LIN {X 0,Y 496.751,Z 364.923,A -85,B 0,C 180,E1 23860.178,E2 23860.178} C_VEL
LIN {X 0,Y 496.699,Z 364.922,A -85,B 0,C 180,E1 23856.821,E2 23856.821} C_VEL
LIN {X 0,Y 496.696,Z 364.92,A -85,B 0,C 180,E1 23853.178,E2 23853.178} C_VEL
LIN {X 0,Y 496.745,Z 364.921,A -85,B 0,C 180,E1 23849.769,E2 23849.769} C_VEL
LIN {X 0,Y 496.722,Z 364.92,A -85,B 0,C 180,E1 23846.307,E2 23846.307} C_VEL
LIN {X 0,Y 496.696,Z 364.92,A -85,B 0,C 180,E1 23842.943,E2 23842.943} C_VEL
LIN {X 0,Y 496.732,Z 364.923,A -85,B 0,C 180,E1 23839.563,E2 23839.563} C_VEL
LIN {X 0,Y 496.727,Z 364.921,A -85,B 0,C 180,E1 23836.141,E2 23836.141} C_VEL
LIN {X 0,Y 496.694,Z 364.922,A -85,B 0,C 180,E1 23832.787,E2 23832.787} C_VEL
LIN {X 0,Y 496.723,Z 364.923,A -85,B 0,C 180,E1 23829.374,E2 23829.374} C_VEL
LIN {X 0,Y 496.725,Z 364.922,A -85,B 0,C 180,E1 23826.045,E2 23826.045} C_VEL
LIN {X 0,Y 496.693,Z 364.922,A -85,B 0,C 180,E1 23822.592,E2 23822.592} C_VEL
LIN {X 0,Y 496.711,Z 364.924,A -85,B 0,C 180,E1 23819.116,E2 23819.116} C_VEL
LIN {X 0,Y 496.752,Z 364.924,A -85,B 0,C 180,E1 23815.696,E2 23815.696} C_VEL
LIN {X 0,Y 496.697,Z 364.925,A -85,B 0,C 180,E1 23812.269,E2 23812.269} C_VEL
LIN {X 0,Y 496.694,Z 364.923,A -85,B 0,C 180,E1 23808.679,E2 23808.679} C_VEL
LIN {X 0,Y 496.739,Z 364.924,A -85,B 0,C 180,E1 23805.279,E2 23805.279} C_VEL
LIN {X 0,Y 496.717,Z 364.924,A -85,B 0,C 180,E1 23801.859,E2 23801.859} C_VEL
LIN {X 0,Y 496.691,Z 364.925,A -85,B 0,C 180,E1 23798.457,E2 23798.457} C_VEL
LIN {X 0,Y 496.723,Z 364.926,A -85,B 0,C 180,E1 23795.007,E2 23795.007} C_VEL
LIN {X 0,Y 496.737,Z 364.925,A -85,B 0,C 180,E1 23791.557,E2 23791.557} C_VEL
LIN {X 0,Y 496.735,Z 365.024,A -85,B 0,C 180,E1 23790.965,E2 23790.965} C_VEL
LIN {X 0,Y 501.684,Z 383.717,A -85,B 0,C 180,E1 23788.187,E2 23788.187} C_VEL
LIN {X 0,Y 500.546,Z 410.556,A -85,B 0,C 180,E1 23784.802,E2 23784.802} C_VEL
LIN {X 0,Y 499.492,Z 438.729,A -85,B 0,C 180,E1 23781.304,E2 23781.304} C_VEL
LIN {X 0,Y 498.454,Z 468.768,A -85,B 0,C 180,E1 23777.632,E2 23777.632} C_VEL
LIN {X 0,Y 498.176,Z 480.291,A -85,B 0,C 180,E1 23776.272,E2 23776.272} C_VEL
LIN {X 0,Y 499.98,Z 493.845,A -85,B 0,C 180,E1 23775.974,E2 23775.974} C_VEL
LIN {X 0,Y 498.863,Z 596.511,A -85,B 0,C 180,E1 23774.304,E2 23774.304} C_VEL
LIN {X 0,Y 498.66,Z 611.149,A -85,B 0,C 180,E1 23773.864,E2 23773.864} C_VEL
LIN {X 0,Y 498.343,Z 626.502,A -85,B 0,C 180,E1 23773.163,E2 23773.163} C_VEL
LIN {X 0,Y 497.924,Z 640.34,A -85,B 0,C 180,E1 23772.29,E2 23772.29} C_VEL
LIN {X 0,Y 497.546,Z 652.64,A -85,B 0,C 180,E1 23771.28,E2 23771.28} C_VEL
LIN {X 0,Y 497.197,Z 664.163,A -85,B 0,C 180,E1 23770.076,E2 23770.076} C_VEL
LIN {X 0,Y 496.862,Z 674.559,A -85,B 0,C 180,E1 23768.681,E2 23768.681} C_VEL
LIN {X 0,Y 496.633,Z 682.68,A -85,B 0,C 180,E1 23767.287,E2 23767.287} C_VEL
LIN {X 0,Y 496.463,Z 689.464,A -85,B 0,C 180,E1 23765.78,E2 23765.78} C_VEL
LIN {X 0,Y 496.36,Z 694.745,A -85,B 0,C 180,E1 23764.159,E2 23764.159} C_VEL
LIN {X 0,Y 496.314,Z 698.292,A -85,B 0,C 180,E1 23762.54,E2 23762.54} C_VEL
LIN {X 0,Y 496.314,Z 700.303,A -85,B 0,C 180,E1 23760.693,E2 23760.693} C_VEL
LIN {X 0,Y 496.325,Z 700.295,A -85,B 0,C 180,E1 23758.961,E2 23758.961} C_VEL
LIN {X 0,Y 496.378,Z 698.701,A -85,B 0,C 180,E1 23757.345,E2 23757.345} C_VEL
LIN {X 0,Y 496.477,Z 695.115,A -85,B 0,C 180,E1 23755.611,E2 23755.611} C_VEL
LIN {X 0,Y 496.626,Z 689.899,A -85,B 0,C 180,E1 23753.991,E2 23753.991} C_VEL
LIN {X 0,Y 496.84,Z 683.239,A -85,B 0,C 180,E1 23752.484,E2 23752.484} C_VEL
LIN {X 0,Y 497.137,Z 674.143,A -85,B 0,C 180,E1 23750.94,E2 23750.94} C_VEL
LIN {X 0,Y 497.497,Z 664.083,A -85,B 0,C 180,E1 23749.62,E2 23749.62} C_VEL
LIN {X 0,Y 497.881,Z 653.043,A -85,B 0,C 180,E1 23748.474,E2 23748.474} C_VEL
LIN {X 0,Y 498.288,Z 640.076,A -85,B 0,C 180,E1 23747.425,E2 23747.425} C_VEL
LIN {X 0,Y 498.681,Z 626.863,A -85,B 0,C 180,E1 23746.61,E2 23746.61} C_VEL
LIN {X 0,Y 499.001,Z 612.986,A -85,B 0,C 180,E1 23745.969,E2 23745.969} C_VEL
LIN {X 0,Y 499.261,Z 596.561,A -85,B 0,C 180,E1 23745.466,E2 23745.466} C_VEL
LIN {X 0,Y 501.106,Z 491.5,A -85,B 0,C 180,E1 23743.486,E2 23743.486} C_VEL
LIN {X 0,Y 498.994,Z 479.897,A -85,B 0,C 180,E1 23743.11,E2 23743.11} C_VEL
LIN {X 0,Y 500.287,Z 449.814,A -85,B 0,C 180,E1 23739.345,E2 23739.345} C_VEL
LIN {X 0,Y 501.876,Z 420.998,A -85,B 0,C 180,E1 23735.645,E2 23735.645} C_VEL
LIN {X 0,Y 503.631,Z 394.385,A -85,B 0,C 180,E1 23732.125,E2 23732.125} C_VEL
LIN {X 0,Y 503.952,Z 388.255,A -85,B 0,C 180,E1 23731.277,E2 23731.277} C_VEL
LIN {X 0,Y 500.616,Z 376.388,A -85,B 0,C 180,E1 23729.185,E2 23729.185} C_VEL
LIN {X 0,Y 497.744,Z 368.01,A -85,B 0,C 180,E1 23727.532,E2 23727.532} C_VEL
LIN {X 0,Y 496.733,Z 364.926,A -85,B 0,C 180,E1 23726.862,E2 23726.862} C_VEL
LIN {X 0,Y 496.695,Z 364.928,A -85,B 0,C 180,E1 23723.426,E2 23723.426} C_VEL
LIN {X 0,Y 496.705,Z 364.927,A -85,B 0,C 180,E1 23719.898,E2 23719.898} C_VEL
LIN {X 0,Y 496.754,Z 364.923,A -85,B 0,C 180,E1 23716.499,E2 23716.499} C_VEL
LIN {X 0,Y 496.707,Z 364.927,A -85,B 0,C 180,E1 23713.032,E2 23713.032} C_VEL
LIN {X 0,Y 496.698,Z 364.929,A -85,B 0,C 180,E1 23709.558,E2 23709.558} C_VEL
LIN {X 0,Y 496.731,Z 364.976,A -85,B 0,C 180,E1 23706.762,E2 23706.762} C_VEL
LIN {X 0,Y 501.559,Z 377.294,A -85,B 0,C 180,E1 23704.76,E2 23704.76} C_VEL
LIN {X 0,Y 505.972,Z 390.476,A -85,B 0,C 180,E1 23702.98,E2 23702.98} C_VEL
LIN {X 0,Y 506.201,Z 393.068,A -85,B 0,C 180,E1 23702.707,E2 23702.707} C_VEL
LIN {X 0,Y 503.796,Z 428.513,A -85,B 0,C 180,E1 23699.616,E2 23699.616} C_VEL
LIN {X 0,Y 502.352,Z 459.871,A -85,B 0,C 180,E1 23697.072,E2 23697.072} C_VEL
LIN {X 0,Y 504.653,Z 479.011,A -85,B 0,C 180,E1 23696.617,E2 23696.617} C_VEL
LIN {X 0,Y 502.285,Z 671.543,A -85,B 0,C 180,E1 23693.566,E2 23693.566} C_VEL
LIN {X 0,Y 501.774,Z 690.29,A -85,B 0,C 180,E1 23693.063,E2 23693.063} C_VEL
LIN {X 0,Y 501.171,Z 707.716,A -85,B 0,C 180,E1 23692.399,E2 23692.399} C_VEL
LIN {X 0,Y 500.457,Z 725.455,A -85,B 0,C 180,E1 23691.507,E2 23691.507} C_VEL
LIN {X 0,Y 499.694,Z 742.452,A -85,B 0,C 180,E1 23690.425,E2 23690.425} C_VEL
LIN {X 0,Y 498.903,Z 758.968,A -85,B 0,C 180,E1 23689.128,E2 23689.128} C_VEL
LIN {X 0,Y 498.093,Z 776.364,A -85,B 0,C 180,E1 23687.464,E2 23687.464} C_VEL
LIN {X 0,Y 497.466,Z 790.207,A -85,B 0,C 180,E1 23685.864,E2 23685.864} C_VEL
LIN {X 0,Y 496.95,Z 802.925,A -85,B 0,C 180,E1 23684.09,E2 23684.09} C_VEL
LIN {X 0,Y 496.554,Z 814.06,A -85,B 0,C 180,E1 23682.206,E2 23682.206} C_VEL
LIN {X 0,Y 496.27,Z 823.123,A -85,B 0,C 180,E1 23680.33,E2 23680.33} C_VEL
LIN {X 0,Y 496.103,Z 830.766,A -85,B 0,C 180,E1 23678.344,E2 23678.344} C_VEL
LIN {X 0,Y 495.998,Z 836.603,A -85,B 0,C 180,E1 23676.366,E2 23676.366} C_VEL
LIN {X 0,Y 495.942,Z 840.96,A -85,B 0,C 180,E1 23674.278,E2 23674.278} C_VEL
LIN {X 0,Y 495.928,Z 843.567,A -85,B 0,C 180,E1 23672.195,E2 23672.195} C_VEL
LIN {X 0,Y 495.93,Z 844.497,A -85,B 0,C 180,E1 23670,E2 23670} C_VEL
LIN {X 0,Y 495.928,Z 843.574,A -85,B 0,C 180,E1 23667.805,E2 23667.805} C_VEL
LIN {X 0,Y 495.94,Z 840.986,A -85,B 0,C 180,E1 23665.722,E2 23665.722} C_VEL
LIN {X 0,Y 495.994,Z 836.643,A -85,B 0,C 180,E1 23663.628,E2 23663.628} C_VEL
LIN {X 0,Y 496.101,Z 830.493,A -85,B 0,C 180,E1 23661.539,E2 23661.539} C_VEL
LIN {X 0,Y 496.28,Z 822.486,A -85,B 0,C 180,E1 23659.475,E2 23659.475} C_VEL
LIN {X 0,Y 496.582,Z 813.139,A -85,B 0,C 180,E1 23657.558,E2 23657.558} C_VEL
LIN {X 0,Y 497.007,Z 801.856,A -85,B 0,C 180,E1 23655.673,E2 23655.673} C_VEL
LIN {X 0,Y 497.572,Z 788.991,A -85,B 0,C 180,E1 23653.9,E2 23653.9} C_VEL
LIN {X 0,Y 498.237,Z 775.03,A -85,B 0,C 180,E1 23652.3,E2 23652.3} C_VEL
LIN {X 0,Y 498.965,Z 760.111,A -85,B 0,C 180,E1 23650.875,E2 23650.875} C_VEL
LIN {X 0,Y 499.76,Z 743.736,A -85,B 0,C 180,E1 23649.583,E2 23649.583} C_VEL
LIN {X 0,Y 500.53,Z 726.786,A -85,B 0,C 180,E1 23648.496,E2 23648.496} C_VEL
LIN {X 0,Y 501.249,Z 709.283,A -85,B 0,C 180,E1 23647.605,E2 23647.605} C_VEL
LIN {X 0,Y 501.911,Z 690.523,A -85,B 0,C 180,E1 23646.882,E2 23646.882} C_VEL
LIN {X 0,Y 502.427,Z 671.773,A -85,B 0,C 180,E1 23646.379,E2 23646.379} C_VEL
LIN {X 0,Y 502.791,Z 638.461,A -85,B 0,C 180,E1 23645.851,E2 23645.851} C_VEL
LIN {X 0,Y 504.288,Z 488.771,A -85,B 0,C 180,E1 23643.587,E2 23643.587} C_VEL
LIN {X 0,Y 504.3,Z 475.833,A -85,B 0,C 180,E1 23643.348,E2 23643.348} C_VEL
LIN {X 0,Y 502.499,Z 461.039,A -85,B 0,C 180,E1 23642.946,E2 23642.946} C_VEL
LIN {X 0,Y 504.592,Z 415.262,A -85,B 0,C 180,E1 23639.254,E2 23639.254} C_VEL
LIN {X 0,Y 505.68,Z 390.578,A -85,B 0,C 180,E1 23637.196,E2 23637.196} C_VEL
LIN {X 0,Y 497.568,Z 367.691,A -85,B 0,C 180,E1 23634.572,E2 23634.572} C_VEL
LIN {X 0,Y 496.708,Z 364.925,A -85,B 0,C 180,E1 23634.216,E2 23634.216} C_VEL
LIN {X 0,Y 496.698,Z 364.926,A -85,B 0,C 180,E1 23630.796,E2 23630.796} C_VEL
LIN {X 0,Y 496.75,Z 364.923,A -85,B 0,C 180,E1 23627.444,E2 23627.444} C_VEL
LIN {X 0,Y 496.717,Z 364.926,A -85,B 0,C 180,E1 23623.984,E2 23623.984} C_VEL
LIN {X 0,Y 496.693,Z 364.926,A -85,B 0,C 180,E1 23620.557,E2 23620.557} C_VEL
LIN {X 0,Y 496.729,Z 364.926,A -85,B 0,C 180,E1 23617.145,E2 23617.145} C_VEL
LIN {X 0,Y 496.725,Z 364.928,A -85,B 0,C 180,E1 23613.749,E2 23613.749} C_VEL
LIN {X 0,Y 496.733,Z 365.09,A -85,B 0,C 180,E1 23611.877,E2 23611.877} C_VEL
LIN {X 0,Y 502.332,Z 381.373,A -85,B 0,C 180,E1 23609.918,E2 23609.918} C_VEL
LIN {X 0,Y 504.151,Z 388.316,A -85,B 0,C 180,E1 23609.136,E2 23609.136} C_VEL
LIN {X 0,Y 503.782,Z 409.778,A -85,B 0,C 180,E1 23607.21,E2 23607.21} C_VEL
LIN {X 0,Y 505.798,Z 422.143,A -85,B 0,C 180,E1 23606.837,E2 23606.837} C_VEL
LIN {X 0,Y 503.551,Z 543.564,A -85,B 0,C 180,E1 23604.775,E2 23604.775} C_VEL
LIN {X 0,Y 502.661,Z 617.661,A -85,B 0,C 180,E1 23603.578,E2 23603.578} C_VEL
LIN {X 0,Y 502.231,Z 637.007,A -85,B 0,C 180,E1 23603.045,E2 23603.045} C_VEL
LIN {X 0,Y 501.643,Z 655.449,A -85,B 0,C 180,E1 23602.315,E2 23602.315} C_VEL
LIN {X 0,Y 500.959,Z 672.625,A -85,B 0,C 180,E1 23601.423,E2 23601.423} C_VEL
LIN {X 0,Y 500.205,Z 689.014,A -85,B 0,C 180,E1 23600.353,E2 23600.353} C_VEL
LIN {X 0,Y 499.419,Z 704.671,A -85,B 0,C 180,E1 23599.096,E2 23599.096} C_VEL
LIN {X 0,Y 498.61,Z 719.701,A -85,B 0,C 180,E1 23597.626,E2 23597.626} C_VEL
LIN {X 0,Y 497.909,Z 732.715,A -85,B 0,C 180,E1 23596.088,E2 23596.088} C_VEL
LIN {X 0,Y 497.261,Z 745.111,A -85,B 0,C 180,E1 23594.319,E2 23594.319} C_VEL
LIN {X 0,Y 496.775,Z 755.393,A -85,B 0,C 180,E1 23592.535,E2 23592.535} C_VEL
LIN {X 0,Y 496.395,Z 764.643,A -85,B 0,C 180,E1 23590.562,E2 23590.562} C_VEL
LIN {X 0,Y 496.155,Z 772.012,A -85,B 0,C 180,E1 23588.576,E2 23588.576} C_VEL
LIN {X 0,Y 496.012,Z 777.934,A -85,B 0,C 180,E1 23586.481,E2 23586.481} C_VEL
LIN {X 0,Y 495.949,Z 782.094,A -85,B 0,C 180,E1 23584.394,E2 23584.394} C_VEL
LIN {X 0,Y 495.931,Z 784.724,A -85,B 0,C 180,E1 23582.195,E2 23582.195} C_VEL
LIN {X 0,Y 495.93,Z 785.607,A -85,B 0,C 180,E1 23580,E2 23580} C_VEL
LIN {X 0,Y 495.927,Z 784.755,A -85,B 0,C 180,E1 23577.805,E2 23577.805} C_VEL
LIN {X 0,Y 495.946,Z 782.175,A -85,B 0,C 180,E1 23575.606,E2 23575.606} C_VEL
LIN {X 0,Y 496.007,Z 778.067,A -85,B 0,C 180,E1 23573.518,E2 23573.518} C_VEL
LIN {X 0,Y 496.138,Z 772.194,A -85,B 0,C 180,E1 23571.423,E2 23571.423} C_VEL
LIN {X 0,Y 496.368,Z 764.816,A -85,B 0,C 180,E1 23569.423,E2 23569.423} C_VEL
LIN {X 0,Y 496.738,Z 755.595,A -85,B 0,C 180,E1 23567.444,E2 23567.444} C_VEL
LIN {X 0,Y 497.252,Z 744.768,A -85,B 0,C 180,E1 23565.562,E2 23565.562} C_VEL
LIN {X 0,Y 497.909,Z 732.382,A -85,B 0,C 180,E1 23563.792,E2 23563.792} C_VEL
LIN {X 0,Y 498.693,Z 718.34,A -85,B 0,C 180,E1 23562.136,E2 23562.136} C_VEL
LIN {X 0,Y 499.508,Z 703.773,A -85,B 0,C 180,E1 23560.714,E2 23560.714} C_VEL
LIN {X 0,Y 500.33,Z 688.341,A -85,B 0,C 180,E1 23559.468,E2 23559.468} C_VEL
LIN {X 0,Y 501.139,Z 672.097,A -85,B 0,C 180,E1 23558.397,E2 23558.397} C_VEL
LIN {X 0,Y 501.883,Z 655.312,A -85,B 0,C 180,E1 23557.511,E2 23557.511} C_VEL
LIN {X 0,Y 502.537,Z 636.894,A -85,B 0,C 180,E1 23556.765,E2 23556.765} C_VEL
LIN {X 0,Y 503.041,Z 617.958,A -85,B 0,C 180,E1 23556.222,E2 23556.222} C_VEL
LIN {X 0,Y 503.395,Z 592.619,A -85,B 0,C 180,E1 23555.783,E2 23555.783} C_VEL
LIN {X 0,Y 505.661,Z 420.696,A -85,B 0,C 180,E1 23553.073,E2 23553.073} C_VEL
LIN {X 0,Y 504.059,Z 412.019,A -85,B 0,C 180,E1 23552.83,E2 23552.83} C_VEL
LIN {X 0,Y 503.132,Z 407.014,A -85,B 0,C 180,E1 23552.598,E2 23552.598} C_VEL
LIN {X 0,Y 501.689,Z 400.932,A -85,B 0,C 180,E1 23552.074,E2 23552.074} C_VEL
LIN {X 0,Y 498.85,Z 394.215,A -85,B 0,C 180,E1 23551.252,E2 23551.252} C_VEL
LIN {X 0,Y 495.123,Z 386.112,A -85,B 0,C 180,E1 23550.212,E2 23550.212} C_VEL
LIN {X 0,Y 488.761,Z 365.913,A -85,B 0,C 180,E1 23547.763,E2 23547.763} C_VEL
LIN {X 0,Y 488.803,Z 365.91,A -85,B 0,C 180,E1 23544.34,E2 23544.34} C_VEL
LIN {X 0,Y 488.793,Z 365.913,A -85,B 0,C 180,E1 23540.83,E2 23540.83} C_VEL
LIN {X 0,Y 488.759,Z 365.913,A -85,B 0,C 180,E1 23537.38,E2 23537.38} C_VEL
LIN {X 0,Y 488.776,Z 365.913,A -85,B 0,C 180,E1 23533.906,E2 23533.906} C_VEL
LIN {X 0,Y 488.826,Z 365.911,A -85,B 0,C 180,E1 23530.422,E2 23530.422} C_VEL
LIN {X 0,Y 488.769,Z 365.912,A -85,B 0,C 180,E1 23526.972,E2 23526.972} C_VEL
LIN {X 0,Y 488.758,Z 365.913,A -85,B 0,C 180,E1 23523.388,E2 23523.388} C_VEL
LIN {X 0,Y 488.789,Z 365.911,A -85,B 0,C 180,E1 23519.942,E2 23519.942} C_VEL
LIN {X 0,Y 488.8,Z 365.911,A -85,B 0,C 180,E1 23516.483,E2 23516.483} C_VEL
LIN {X 0,Y 488.758,Z 365.911,A -85,B 0,C 180,E1 23513.128,E2 23513.128} C_VEL
LIN {X 0,Y 488.771,Z 365.912,A -85,B 0,C 180,E1 23509.602,E2 23509.602} C_VEL
LIN {X 0,Y 488.818,Z 365.91,A -85,B 0,C 180,E1 23506.152,E2 23506.152} C_VEL
LIN {X 0,Y 488.764,Z 365.909,A -85,B 0,C 180,E1 23502.764,E2 23502.764} C_VEL
LIN {X 0,Y 488.758,Z 365.909,A -85,B 0,C 180,E1 23499.182,E2 23499.182} C_VEL
LIN {X 0,Y 488.795,Z 365.911,A -85,B 0,C 180,E1 23495.753,E2 23495.753} C_VEL
LIN {X 0,Y 488.798,Z 365.908,A -85,B 0,C 180,E1 23492.227,E2 23492.227} C_VEL
LIN {X 0,Y 488.755,Z 365.909,A -85,B 0,C 180,E1 23488.828,E2 23488.828} C_VEL
LIN {X 0,Y 488.766,Z 365.912,A -85,B 0,C 180,E1 23485.306,E2 23485.306} C_VEL
LIN {X 0,Y 488.82,Z 365.908,A -85,B 0,C 180,E1 23481.886,E2 23481.886} C_VEL
LIN {X 0,Y 488.767,Z 365.911,A -85,B 0,C 180,E1 23478.435,E2 23478.435} C_VEL
LIN {X 0,Y 488.757,Z 365.912,A -85,B 0,C 180,E1 23474.924,E2 23474.924} C_VEL
LIN {X 0,Y 488.798,Z 365.913,A -85,B 0,C 180,E1 23471.515,E2 23471.515} C_VEL
LIN {X 0,Y 488.792,Z 365.911,A -85,B 0,C 180,E1 23468.016,E2 23468.016} C_VEL
LIN {X 0,Y 488.756,Z 365.911,A -85,B 0,C 180,E1 23464.558,E2 23464.558} C_VEL
LIN {X 0,Y 488.764,Z 365.911,A -85,B 0,C 180,E1 23460.999,E2 23460.999} C_VEL
LIN {X 0,Y 488.815,Z 365.913,A -85,B 0,C 180,E1 23457.594,E2 23457.594} C_VEL
LIN {X 0,Y 488.769,Z 365.914,A -85,B 0,C 180,E1 23454.105,E2 23454.105} C_VEL
LIN {X 0,Y 488.754,Z 365.914,A -85,B 0,C 180,E1 23450.641,E2 23450.641} C_VEL
LIN {X 0,Y 488.792,Z 365.913,A -85,B 0,C 180,E1 23447.224,E2 23447.224} C_VEL
LIN {X 0,Y 488.792,Z 365.912,A -85,B 0,C 180,E1 23443.742,E2 23443.742} C_VEL
LIN {X 0,Y 488.753,Z 365.914,A -85,B 0,C 180,E1 23440.429,E2 23440.429} C_VEL
LIN {X 0,Y 488.778,Z 365.915,A -85,B 0,C 180,E1 23436.972,E2 23436.972} C_VEL
LIN {X 0,Y 488.803,Z 365.913,A -85,B 0,C 180,E1 23433.525,E2 23433.525} C_VEL
LIN {X 0,Y 488.825,Z 365.983,A -85,B 0,C 180,E1 23431.37,E2 23431.37} C_VEL
LIN {X 0,Y 494.13,Z 386.139,A -85,B 0,C 180,E1 23428.331,E2 23428.331} C_VEL
LIN {X 0,Y 492.901,Z 412.749,A -85,B 0,C 180,E1 23424.94,E2 23424.94} C_VEL
LIN {X 0,Y 491.739,Z 441.369,A -85,B 0,C 180,E1 23421.344,E2 23421.344} C_VEL
LIN {X 0,Y 490.645,Z 470.992,A -85,B 0,C 180,E1 23417.676,E2 23417.676} C_VEL
LIN {X 0,Y 490.413,Z 480.136,A -85,B 0,C 180,E1 23416.585,E2 23416.585} C_VEL
LIN {X 0,Y 492.381,Z 494.563,A -85,B 0,C 180,E1 23416.255,E2 23416.255} C_VEL
LIN {X 0,Y 491.147,Z 597.02,A -85,B 0,C 180,E1 23414.543,E2 23414.543} C_VEL
LIN {X 0,Y 490.926,Z 611.877,A -85,B 0,C 180,E1 23414.086,E2 23414.086} C_VEL
LIN {X 0,Y 490.587,Z 627.214,A -85,B 0,C 180,E1 23413.375,E2 23413.375} C_VEL
LIN {X 0,Y 490.144,Z 641.081,A -85,B 0,C 180,E1 23412.488,E2 23412.488} C_VEL
LIN {X 0,Y 489.748,Z 653.15,A -85,B 0,C 180,E1 23411.488,E2 23411.488} C_VEL
LIN {X 0,Y 489.363,Z 665.003,A -85,B 0,C 180,E1 23410.239,E2 23410.239} C_VEL
LIN {X 0,Y 489.002,Z 675.466,A -85,B 0,C 180,E1 23408.821,E2 23408.821} C_VEL
LIN {X 0,Y 488.751,Z 683.637,A -85,B 0,C 180,E1 23407.405,E2 23407.405} C_VEL
LIN {X 0,Y 488.567,Z 690.486,A -85,B 0,C 180,E1 23405.873,E2 23405.873} C_VEL
LIN {X 0,Y 488.452,Z 695.822,A -85,B 0,C 180,E1 23404.226,E2 23404.226} C_VEL
LIN {X 0,Y 488.4,Z 699.416,A -85,B 0,C 180,E1 23402.582,E2 23402.582} C_VEL
LIN {X 0,Y 488.4,Z 701.472,A -85,B 0,C 180,E1 23400.704,E2 23400.704} C_VEL
LIN {X 0,Y 488.417,Z 701.497,A -85,B 0,C 180,E1 23398.944,E2 23398.944} C_VEL
LIN {X 0,Y 488.48,Z 699.899,A -85,B 0,C 180,E1 23397.293,E2 23397.293} C_VEL
LIN {X 0,Y 488.592,Z 696.336,A -85,B 0,C 180,E1 23395.54,E2 23395.54} C_VEL
LIN {X 0,Y 488.762,Z 691.122,A -85,B 0,C 180,E1 23393.894,E2 23393.894} C_VEL
LIN {X 0,Y 489.002,Z 684.46,A -85,B 0,C 180,E1 23392.363,E2 23392.363} C_VEL
LIN {X 0,Y 489.322,Z 675.59,A -85,B 0,C 180,E1 23390.829,E2 23390.829} C_VEL
LIN {X 0,Y 489.714,Z 665.44,A -85,B 0,C 180,E1 23389.471,E2 23389.471} C_VEL
LIN {X 0,Y 490.133,Z 654.283,A -85,B 0,C 180,E1 23388.292,E2 23388.292} C_VEL
LIN {X 0,Y 490.58,Z 640.988,A -85,B 0,C 180,E1 23387.201,E2 23387.201} C_VEL
LIN {X 0,Y 491.017,Z 627.095,A -85,B 0,C 180,E1 23386.337,E2 23386.337} C_VEL
LIN {X 0,Y 491.367,Z 612.611,A -85,B 0,C 180,E1 23385.671,E2 23385.671} C_VEL
LIN {X 0,Y 491.64,Z 596.868,A -85,B 0,C 180,E1 23385.186,E2 23385.186} C_VEL
LIN {X 0,Y 493.774,Z 492.682,A -85,B 0,C 180,E1 23383.128,E2 23383.128} C_VEL
LIN {X 0,Y 491.446,Z 479.838,A -85,B 0,C 180,E1 23382.69,E2 23382.69} C_VEL
LIN {X 0,Y 492.86,Z 450.417,A -85,B 0,C 180,E1 23378.94,E2 23378.94} C_VEL
LIN {X 0,Y 494.579,Z 422.271,A -85,B 0,C 180,E1 23375.262,E2 23375.262} C_VEL
LIN {X 0,Y 496.628,Z 395.455,A -85,B 0,C 180,E1 23371.632,E2 23371.632} C_VEL
LIN {X 0,Y 496.867,Z 391.627,A -85,B 0,C 180,E1 23371.089,E2 23371.089} C_VEL
LIN {X 0,Y 493.795,Z 380.405,A -85,B 0,C 180,E1 23369.049,E2 23369.049} C_VEL
LIN {X 0,Y 490.962,Z 372.107,A -85,B 0,C 180,E1 23367.338,E2 23367.338} C_VEL
LIN {X 0,Y 488.763,Z 365.918,A -85,B 0,C 180,E1 23365.908,E2 23365.908} C_VEL
LIN {X 0,Y 488.812,Z 365.912,A -85,B 0,C 180,E1 23362.443,E2 23362.443} C_VEL
LIN {X 0,Y 488.774,Z 365.916,A -85,B 0,C 180,E1 23359.012,E2 23359.012} C_VEL
LIN {X 0,Y 488.755,Z 365.917,A -85,B 0,C 180,E1 23355.558,E2 23355.558} C_VEL
LIN {X 0,Y 488.795,Z 365.915,A -85,B 0,C 180,E1 23352.14,E2 23352.14} C_VEL
LIN {X 0,Y 488.786,Z 365.913,A -85,B 0,C 180,E1 23348.752,E2 23348.752} C_VEL
LIN {X 0,Y 488.774,Z 365.982,A -85,B 0,C 180,E1 23347.709,E2 23347.709} C_VEL
LIN {X 0,Y 489.998,Z 369.292,A -85,B 0,C 180,E1 23347.075,E2 23347.075} C_VEL
LIN {X 0,Y 493.352,Z 377.235,A -85,B 0,C 180,E1 23345.64,E2 23345.64} C_VEL
LIN {X 0,Y 497.269,Z 388.206,A -85,B 0,C 180,E1 23343.985,E2 23343.985} C_VEL
LIN {X 0,Y 499.212,Z 395.195,A -85,B 0,C 180,E1 23343.079,E2 23343.079} C_VEL
LIN {X 0,Y 496.611,Z 428.436,A -85,B 0,C 180,E1 23340.088,E2 23340.088} C_VEL
LIN {X 0,Y 494.953,Z 459.203,A -85,B 0,C 180,E1 23337.515,E2 23337.515} C_VEL
LIN {X 0,Y 497.452,Z 480.045,A -85,B 0,C 180,E1 23337.005,E2 23337.005} C_VEL
LIN {X 0,Y 494.818,Z 671.2,A -85,B 0,C 180,E1 23333.904,E2 23333.904} C_VEL
LIN {X 0,Y 494.249,Z 690.099,A -85,B 0,C 180,E1 23333.388,E2 23333.388} C_VEL
LIN {X 0,Y 493.572,Z 708.044,A -85,B 0,C 180,E1 23332.687,E2 23332.687} C_VEL
LIN {X 0,Y 492.808,Z 725.396,A -85,B 0,C 180,E1 23331.795,E2 23331.795} C_VEL
LIN {X 0,Y 491.988,Z 742.176,A -85,B 0,C 180,E1 23330.709,E2 23330.709} C_VEL
LIN {X 0,Y 491.123,Z 758.792,A -85,B 0,C 180,E1 23329.381,E2 23329.381} C_VEL
LIN {X 0,Y 490.32,Z 774.264,A -85,B 0,C 180,E1 23327.873,E2 23327.873} C_VEL
LIN {X 0,Y 489.618,Z 788.077,A -85,B 0,C 180,E1 23326.247,E2 23326.247} C_VEL
LIN {X 0,Y 489.035,Z 800.776,A -85,B 0,C 180,E1 23324.444,E2 23324.444} C_VEL
LIN {X 0,Y 488.574,Z 813.256,A -85,B 0,C 180,E1 23322.289,E2 23322.289} C_VEL
LIN {X 0,Y 488.297,Z 822.273,A -85,B 0,C 180,E1 23320.381,E2 23320.381} C_VEL
LIN {X 0,Y 488.143,Z 829.875,A -85,B 0,C 180,E1 23318.362,E2 23318.362} C_VEL
LIN {X 0,Y 488.054,Z 835.662,A -85,B 0,C 180,E1 23316.352,E2 23316.352} C_VEL
LIN {X 0,Y 488.011,Z 839.964,A -85,B 0,C 180,E1 23314.23,E2 23314.23} C_VEL
LIN {X 0,Y 488.005,Z 842.518,A -85,B 0,C 180,E1 23312.114,E2 23312.114} C_VEL
LIN {X 0,Y 488.008,Z 843.381,A -85,B 0,C 180,E1 23310,E2 23310} C_VEL
LIN {X 0,Y 488,Z 842.559,A -85,B 0,C 180,E1 23307.886,E2 23307.886} C_VEL
LIN {X 0,Y 488.001,Z 840.056,A -85,B 0,C 180,E1 23305.77,E2 23305.77} C_VEL
LIN {X 0,Y 488.04,Z 835.803,A -85,B 0,C 180,E1 23303.648,E2 23303.648} C_VEL
LIN {X 0,Y 488.129,Z 829.72,A -85,B 0,C 180,E1 23301.519,E2 23301.519} C_VEL
LIN {X 0,Y 488.302,Z 821.636,A -85,B 0,C 180,E1 23299.38,E2 23299.38} C_VEL
LIN {X 0,Y 488.623,Z 811.889,A -85,B 0,C 180,E1 23297.352,E2 23297.352} C_VEL
LIN {X 0,Y 489.071,Z 800.544,A -85,B 0,C 180,E1 23295.436,E2 23295.436} C_VEL
LIN {X 0,Y 489.655,Z 788.005,A -85,B 0,C 180,E1 23293.683,E2 23293.683} C_VEL
LIN {X 0,Y 490.351,Z 774.12,A -85,B 0,C 180,E1 23292.067,E2 23292.067} C_VEL
LIN {X 0,Y 491.132,Z 759.186,A -85,B 0,C 180,E1 23290.619,E2 23290.619} C_VEL
LIN {X 0,Y 491.997,Z 742.558,A -85,B 0,C 180,E1 23289.292,E2 23289.292} C_VEL
LIN {X 0,Y 492.817,Z 725.809,A -85,B 0,C 180,E1 23288.205,E2 23288.205} C_VEL
LIN {X 0,Y 493.614,Z 707.746,A -85,B 0,C 180,E1 23287.278,E2 23287.278} C_VEL
LIN {X 0,Y 494.305,Z 689.146,A -85,B 0,C 180,E1 23286.56,E2 23286.56} C_VEL
LIN {X 0,Y 494.859,Z 670.35,A -85,B 0,C 180,E1 23286.058,E2 23286.058} C_VEL
LIN {X 0,Y 495.371,Z 621.762,A -85,B 0,C 180,E1 23285.3,E2 23285.3} C_VEL
LIN {X 0,Y 496.552,Z 517.237,A -85,B 0,C 180,E1 23283.678,E2 23283.678} C_VEL
LIN {X 0,Y 497.199,Z 477.016,A -85,B 0,C 180,E1 23282.943,E2 23282.943} C_VEL
LIN {X 0,Y 495.1,Z 459.453,A -85,B 0,C 180,E1 23282.445,E2 23282.445} C_VEL
LIN {X 0,Y 497.454,Z 413.121,A -85,B 0,C 180,E1 23278.629,E2 23278.629} C_VEL
LIN {X 0,Y 498.476,Z 393.585,A -85,B 0,C 180,E1 23276.975,E2 23276.975} C_VEL
LIN {X 0,Y 490.645,Z 371.492,A -85,B 0,C 180,E1 23274.4,E2 23274.4} C_VEL
LIN {X 0,Y 488.814,Z 365.911,A -85,B 0,C 180,E1 23273.699,E2 23273.699} C_VEL
LIN {X 0,Y 488.765,Z 365.915,A -85,B 0,C 180,E1 23270.28,E2 23270.28} C_VEL
LIN {X 0,Y 488.758,Z 365.915,A -85,B 0,C 180,E1 23266.739,E2 23266.739} C_VEL
LIN {X 0,Y 488.797,Z 365.913,A -85,B 0,C 180,E1 23263.263,E2 23263.263} C_VEL
LIN {X 0,Y 488.778,Z 365.916,A -85,B 0,C 180,E1 23259.904,E2 23259.904} C_VEL
LIN {X 0,Y 488.754,Z 365.916,A -85,B 0,C 180,E1 23256.488,E2 23256.488} C_VEL
LIN {X 0,Y 488.782,Z 365.919,A -85,B 0,C 180,E1 23252.996,E2 23252.996} C_VEL
LIN {X 0,Y 488.775,Z 366.07,A -85,B 0,C 180,E1 23252.513,E2 23252.513} C_VEL
LIN {X 0,Y 494.273,Z 381.068,A -85,B 0,C 180,E1 23250.611,E2 23250.611} C_VEL
LIN {X 0,Y 497.09,Z 391.58,A -85,B 0,C 180,E1 23249.392,E2 23249.392} C_VEL
LIN {X 0,Y 496.757,Z 410.749,A -85,B 0,C 180,E1 23247.671,E2 23247.671} C_VEL
LIN {X 0,Y 498.795,Z 423.346,A -85,B 0,C 180,E1 23247.265,E2 23247.265} C_VEL
LIN {X 0,Y 496.208,Z 543.735,A -85,B 0,C 180,E1 23245.139,E2 23245.139} C_VEL
LIN {X 0,Y 495.166,Z 618.664,A -85,B 0,C 180,E1 23243.886,E2 23243.886} C_VEL
LIN {X 0,Y 494.688,Z 638.035,A -85,B 0,C 180,E1 23243.334,E2 23243.334} C_VEL
LIN {X 0,Y 494.083,Z 655.925,A -85,B 0,C 180,E1 23242.612,E2 23242.612} C_VEL
LIN {X 0,Y 493.335,Z 673.427,A -85,B 0,C 180,E1 23241.687,E2 23241.687} C_VEL
LIN {X 0,Y 492.507,Z 690.303,A -85,B 0,C 180,E1 23240.562,E2 23240.562} C_VEL
LIN {X 0,Y 491.641,Z 706.391,A -85,B 0,C 180,E1 23239.236,E2 23239.236} C_VEL
LIN {X 0,Y 490.784,Z 721.344,A -85,B 0,C 180,E1 23237.732,E2 23237.732} C_VEL
LIN {X 0,Y 490.017,Z 734.655,A -85,B 0,C 180,E1 23236.111,E2 23236.111} C_VEL
LIN {X 0,Y 489.345,Z 746.845,A -85,B 0,C 180,E1 23234.314,E2 23234.314} C_VEL
LIN {X 0,Y 488.815,Z 757.454,A -85,B 0,C 180,E1 23232.402,E2 23232.402} C_VEL
LIN {X 0,Y 488.42,Z 766.473,A -85,B 0,C 180,E1 23230.378,E2 23230.378} C_VEL
LIN {X 0,Y 488.175,Z 773.558,A -85,B 0,C 180,E1 23228.361,E2 23228.361} C_VEL
LIN {X 0,Y 488.029,Z 779.191,A -85,B 0,C 180,E1 23226.234,E2 23226.234} C_VEL
LIN {X 0,Y 487.963,Z 783.086,A -85,B 0,C 180,E1 23224.112,E2 23224.112} C_VEL
LIN {X 0,Y 487.944,Z 785.357,A -85,B 0,C 180,E1 23221.996,E2 23221.996} C_VEL
LIN {X 0,Y 487.947,Z 786.04,A -85,B 0,C 180,E1 23219.765,E2 23219.765} C_VEL
LIN {X 0,Y 487.945,Z 784.996,A -85,B 0,C 180,E1 23217.534,E2 23217.534} C_VEL
LIN {X 0,Y 487.969,Z 782.399,A -85,B 0,C 180,E1 23215.416,E2 23215.416} C_VEL
LIN {X 0,Y 488.042,Z 778.149,A -85,B 0,C 180,E1 23213.294,E2 23213.294} C_VEL
LIN {X 0,Y 488.196,Z 772.126,A -85,B 0,C 180,E1 23211.164,E2 23211.164} C_VEL
LIN {X 0,Y 488.454,Z 764.657,A -85,B 0,C 180,E1 23209.145,E2 23209.145} C_VEL
LIN {X 0,Y 488.875,Z 755.197,A -85,B 0,C 180,E1 23207.119,E2 23207.119} C_VEL
LIN {X 0,Y 489.451,Z 744.165,A -85,B 0,C 180,E1 23205.205,E2 23205.205} C_VEL
LIN {X 0,Y 490.181,Z 731.545,A -85,B 0,C 180,E1 23203.407,E2 23203.407} C_VEL
LIN {X 0,Y 491.01,Z 717.787,A -85,B 0,C 180,E1 23201.785,E2 23201.785} C_VEL
LIN {X 0,Y 491.899,Z 703.013,A -85,B 0,C 180,E1 23200.342,E2 23200.342} C_VEL
LIN {X 0,Y 492.842,Z 686.524,A -85,B 0,C 180,E1 23199.018,E2 23199.018} C_VEL
LIN {X 0,Y 493.713,Z 669.811,A -85,B 0,C 180,E1 23197.934,E2 23197.934} C_VEL
LIN {X 0,Y 494.535,Z 651.466,A -85,B 0,C 180,E1 23197.001,E2 23197.001} C_VEL
LIN {X 0,Y 495.205,Z 632.791,A -85,B 0,C 180,E1 23196.289,E2 23196.289} C_VEL
LIN {X 0,Y 495.699,Z 613.895,A -85,B 0,C 180,E1 23195.793,E2 23195.793} C_VEL
LIN {X 0,Y 498.414,Z 421.478,A -85,B 0,C 180,E1 23192.668,E2 23192.668} C_VEL
LIN {X 0,Y 495.603,Z 406.34,A -85,B 0,C 180,E1 23192.223,E2 23192.223} C_VEL
LIN {X 0,Y 496.087,Z 389.492,A -85,B 0,C 180,E1 23190.608,E2 23190.608} C_VEL
LIN {X 0,Y 495.123,Z 386.112,A -85,B 0,C 180,E1 23190.212,E2 23190.212} C_VEL
LIN {X 0,Y 493.203,Z 383.008,A -85,B 0,C 180,E1 23189.781,E2 23189.781} C_VEL
LIN {X 0,Y 484.567,Z 376.396,A -85,B 0,C 180,E1 23188.534,E2 23188.534} C_VEL
LIN {X 0,Y 483.183,Z 374.157,A -85,B 0,C 180,E1 23188.216,E2 23188.216} C_VEL
LIN {X 0,Y 480.826,Z 366.903,A -85,B 0,C 180,E1 23187.307,E2 23187.307} C_VEL
LIN {X 0,Y 480.824,Z 366.904,A -85,B 0,C 180,E1 23183.788,E2 23183.788} C_VEL
LIN {X 0,Y 480.866,Z 366.898,A -85,B 0,C 180,E1 23180.295,E2 23180.295} C_VEL
LIN {X 0,Y 480.85,Z 366.901,A -85,B 0,C 180,E1 23176.834,E2 23176.834} C_VEL
LIN {X 0,Y 480.82,Z 366.901,A -85,B 0,C 180,E1 23173.333,E2 23173.333} C_VEL
LIN {X 0,Y 480.834,Z 366.901,A -85,B 0,C 180,E1 23169.827,E2 23169.827} C_VEL
LIN {X 0,Y 480.878,Z 366.901,A -85,B 0,C 180,E1 23166.341,E2 23166.341} C_VEL
LIN {X 0,Y 480.834,Z 366.901,A -85,B 0,C 180,E1 23162.85,E2 23162.85} C_VEL
LIN {X 0,Y 480.819,Z 366.9,A -85,B 0,C 180,E1 23159.389,E2 23159.389} C_VEL
LIN {X 0,Y 480.863,Z 366.901,A -85,B 0,C 180,E1 23156.023,E2 23156.023} C_VEL
LIN {X 0,Y 480.856,Z 366.899,A -85,B 0,C 180,E1 23152.495,E2 23152.495} C_VEL
LIN {X 0,Y 480.821,Z 366.901,A -85,B 0,C 180,E1 23149.055,E2 23149.055} C_VEL
LIN {X 0,Y 480.824,Z 366.902,A -85,B 0,C 180,E1 23145.437,E2 23145.437} C_VEL
LIN {X 0,Y 480.873,Z 366.901,A -85,B 0,C 180,E1 23142.001,E2 23142.001} C_VEL
LIN {X 0,Y 480.841,Z 366.898,A -85,B 0,C 180,E1 23138.49,E2 23138.49} C_VEL
LIN {X 0,Y 480.817,Z 366.899,A -85,B 0,C 180,E1 23135.011,E2 23135.011} C_VEL
LIN {X 0,Y 480.839,Z 366.901,A -85,B 0,C 180,E1 23131.549,E2 23131.549} C_VEL
LIN {X 0,Y 480.868,Z 366.897,A -85,B 0,C 180,E1 23128.093,E2 23128.093} C_VEL
LIN {X 0,Y 480.821,Z 366.9,A -85,B 0,C 180,E1 23124.631,E2 23124.631} C_VEL
LIN {X 0,Y 480.818,Z 366.9,A -85,B 0,C 180,E1 23121.027,E2 23121.027} C_VEL
LIN {X 0,Y 480.85,Z 366.9,A -85,B 0,C 180,E1 23117.511,E2 23117.511} C_VEL
LIN {X 0,Y 480.842,Z 366.901,A -85,B 0,C 180,E1 23114.193,E2 23114.193} C_VEL
LIN {X 0,Y 480.817,Z 366.901,A -85,B 0,C 180,E1 23110.692,E2 23110.692} C_VEL
LIN {X 0,Y 480.827,Z 366.901,A -85,B 0,C 180,E1 23107.103,E2 23107.103} C_VEL
LIN {X 0,Y 480.871,Z 366.9,A -85,B 0,C 180,E1 23103.579,E2 23103.579} C_VEL
LIN {X 0,Y 480.84,Z 366.9,A -85,B 0,C 180,E1 23100.062,E2 23100.062} C_VEL
LIN {X 0,Y 480.815,Z 366.903,A -85,B 0,C 180,E1 23096.559,E2 23096.559} C_VEL
LIN {X 0,Y 480.829,Z 366.904,A -85,B 0,C 180,E1 23092.988,E2 23092.988} C_VEL
LIN {X 0,Y 480.883,Z 366.901,A -85,B 0,C 180,E1 23089.552,E2 23089.552} C_VEL
LIN {X 0,Y 480.831,Z 366.902,A -85,B 0,C 180,E1 23086.01,E2 23086.01} C_VEL
LIN {X 0,Y 480.815,Z 366.903,A -85,B 0,C 180,E1 23082.52,E2 23082.52} C_VEL
LIN {X 0,Y 480.853,Z 366.904,A -85,B 0,C 180,E1 23079.14,E2 23079.14} C_VEL
LIN {X 0,Y 480.855,Z 366.904,A -85,B 0,C 180,E1 23075.607,E2 23075.607} C_VEL
LIN {X 0,Y 480.816,Z 366.907,A -85,B 0,C 180,E1 23072.165,E2 23072.165} C_VEL
LIN {X 0,Y 480.865,Z 367.101,A -85,B 0,C 180,E1 23071.771,E2 23071.771} C_VEL
LIN {X 0,Y 485.935,Z 386.111,A -85,B 0,C 180,E1 23068.849,E2 23068.849} C_VEL
LIN {X 0,Y 486.553,Z 389.639,A -85,B 0,C 180,E1 23068.34,E2 23068.34} C_VEL
LIN {X 0,Y 485.153,Z 417.126,A -85,B 0,C 180,E1 23064.797,E2 23064.797} C_VEL
LIN {X 0,Y 483.864,Z 446.47,A -85,B 0,C 180,E1 23061.073,E2 23061.073} C_VEL
LIN {X 0,Y 482.765,Z 475.164,A -85,B 0,C 180,E1 23057.476,E2 23057.476} C_VEL
LIN {X 0,Y 482.66,Z 479.999,A -85,B 0,C 180,E1 23056.907,E2 23056.907} C_VEL
LIN {X 0,Y 484.793,Z 495.404,A -85,B 0,C 180,E1 23056.544,E2 23056.544} C_VEL
LIN {X 0,Y 483.43,Z 597.711,A -85,B 0,C 180,E1 23054.78,E2 23054.78} C_VEL
LIN {X 0,Y 483.193,Z 612.489,A -85,B 0,C 180,E1 23054.317,E2 23054.317} C_VEL
LIN {X 0,Y 482.84,Z 627.525,A -85,B 0,C 180,E1 23053.611,E2 23053.611} C_VEL
LIN {X 0,Y 482.363,Z 641.757,A -85,B 0,C 180,E1 23052.693,E2 23052.693} C_VEL
LIN {X 0,Y 481.951,Z 653.657,A -85,B 0,C 180,E1 23051.7,E2 23051.7} C_VEL
LIN {X 0,Y 481.53,Z 665.815,A -85,B 0,C 180,E1 23050.408,E2 23050.408} C_VEL
LIN {X 0,Y 481.141,Z 676.346,A -85,B 0,C 180,E1 23048.967,E2 23048.967} C_VEL
LIN {X 0,Y 480.871,Z 684.594,A -85,B 0,C 180,E1 23047.527,E2 23047.527} C_VEL
LIN {X 0,Y 480.67,Z 691.499,A -85,B 0,C 180,E1 23045.97,E2 23045.97} C_VEL
LIN {X 0,Y 480.543,Z 696.894,A -85,B 0,C 180,E1 23044.296,E2 23044.296} C_VEL
LIN {X 0,Y 480.487,Z 700.537,A -85,B 0,C 180,E1 23042.624,E2 23042.624} C_VEL
LIN {X 0,Y 480.488,Z 702.644,A -85,B 0,C 180,E1 23040.716,E2 23040.716} C_VEL
LIN {X 0,Y 480.51,Z 702.7,A -85,B 0,C 180,E1 23038.927,E2 23038.927} C_VEL
LIN {X 0,Y 480.583,Z 701.143,A -85,B 0,C 180,E1 23037.257,E2 23037.257} C_VEL
LIN {X 0,Y 480.712,Z 697.577,A -85,B 0,C 180,E1 23035.467,E2 23035.467} C_VEL
LIN {X 0,Y 480.904,Z 692.363,A -85,B 0,C 180,E1 23033.794,E2 23033.794} C_VEL
LIN {X 0,Y 481.168,Z 685.693,A -85,B 0,C 180,E1 23032.238,E2 23032.238} C_VEL
LIN {X 0,Y 481.519,Z 676.808,A -85,B 0,C 180,E1 23030.679,E2 23030.679} C_VEL
LIN {X 0,Y 481.943,Z 666.665,A -85,B 0,C 180,E1 23029.299,E2 23029.299} C_VEL
LIN {X 0,Y 482.402,Z 655.534,A -85,B 0,C 180,E1 23028.099,E2 23028.099} C_VEL
LIN {X 0,Y 482.905,Z 641.889,A -85,B 0,C 180,E1 23026.957,E2 23026.957} C_VEL
LIN {X 0,Y 483.391,Z 627.596,A -85,B 0,C 180,E1 23026.056,E2 23026.056} C_VEL
LIN {X 0,Y 483.762,Z 613.016,A -85,B 0,C 180,E1 23025.382,E2 23025.382} C_VEL
LIN {X 0,Y 484.049,Z 597.539,A -85,B 0,C 180,E1 23024.899,E2 23024.899} C_VEL
LIN {X 0,Y 486.573,Z 494.289,A -85,B 0,C 180,E1 23022.76,E2 23022.76} C_VEL
LIN {X 0,Y 483.943,Z 479.652,A -85,B 0,C 180,E1 23022.23,E2 23022.23} C_VEL
LIN {X 0,Y 485.489,Z 450.886,A -85,B 0,C 180,E1 23018.495,E2 23018.495} C_VEL
LIN {X 0,Y 487.447,Z 422.347,A -85,B 0,C 180,E1 23014.68,E2 23014.68} C_VEL
LIN {X 0,Y 489.751,Z 396.25,A -85,B 0,C 180,E1 23011.063,E2 23011.063} C_VEL
LIN {X 0,Y 489.493,Z 393.698,A -85,B 0,C 180,E1 23010.644,E2 23010.644} C_VEL
LIN {X 0,Y 486.392,Z 382.25,A -85,B 0,C 180,E1 23008.455,E2 23008.455} C_VEL
LIN {X 0,Y 482.95,Z 372.716,A -85,B 0,C 180,E1 23006.3,E2 23006.3} C_VEL
LIN {X 0,Y 481.613,Z 369.52,A -85,B 0,C 180,E1 23005.475,E2 23005.475} C_VEL
LIN {X 0,Y 480.86,Z 366.902,A -85,B 0,C 180,E1 23004.803,E2 23004.803} C_VEL
LIN {X 0,Y 480.817,Z 366.907,A -85,B 0,C 180,E1 23001.402,E2 23001.402} C_VEL
LIN {X 0,Y 480.822,Z 366.905,A -85,B 0,C 180,E1 22997.757,E2 22997.757} C_VEL
LIN {X 0,Y 480.87,Z 366.902,A -85,B 0,C 180,E1 22994.318,E2 22994.318} C_VEL
LIN {X 0,Y 480.85,Z 366.904,A -85,B 0,C 180,E1 22990.762,E2 22990.762} C_VEL
LIN {X 0,Y 480.843,Z 366.924,A -85,B 0,C 180,E1 22988.825,E2 22988.825} C_VEL
LIN {X 0,Y 482.273,Z 370.557,A -85,B 0,C 180,E1 22988.007,E2 22988.007} C_VEL
LIN {X 0,Y 485.764,Z 378.767,A -85,B 0,C 180,E1 22986.356,E2 22986.356} C_VEL
LIN {X 0,Y 489.725,Z 389.572,A -85,B 0,C 180,E1 22984.582,E2 22984.582} C_VEL
LIN {X 0,Y 492.211,Z 398.103,A -85,B 0,C 180,E1 22983.396,E2 22983.396} C_VEL
LIN {X 0,Y 489.203,Z 432.073,A -85,B 0,C 180,E1 22980.253,E2 22980.253} C_VEL
LIN {X 0,Y 487.615,Z 458.769,A -85,B 0,C 180,E1 22977.969,E2 22977.969} C_VEL
LIN {X 0,Y 490.273,Z 481.182,A -85,B 0,C 180,E1 22977.402,E2 22977.402} C_VEL
LIN {X 0,Y 487.363,Z 671.005,A -85,B 0,C 180,E1 22974.249,E2 22974.249} C_VEL
LIN {X 0,Y 486.742,Z 689.895,A -85,B 0,C 180,E1 22973.722,E2 22973.722} C_VEL
LIN {X 0,Y 486.013,Z 707.809,A -85,B 0,C 180,E1 22973.01,E2 22973.01} C_VEL
LIN {X 0,Y 485.172,Z 725.324,A -85,B 0,C 180,E1 22972.093,E2 22972.093} C_VEL
LIN {X 0,Y 484.285,Z 742.033,A -85,B 0,C 180,E1 22970.99,E2 22970.99} C_VEL
LIN {X 0,Y 483.35,Z 758.604,A -85,B 0,C 180,E1 22969.643,E2 22969.643} C_VEL
LIN {X 0,Y 482.484,Z 774.044,A -85,B 0,C 180,E1 22968.11,E2 22968.11} C_VEL
LIN {X 0,Y 481.746,Z 787.598,A -85,B 0,C 180,E1 22966.489,E2 22966.489} C_VEL
LIN {X 0,Y 481.122,Z 800.119,A -85,B 0,C 180,E1 22964.687,E2 22964.687} C_VEL
LIN {X 0,Y 480.657,Z 811.279,A -85,B 0,C 180,E1 22962.739,E2 22962.739} C_VEL
LIN {X 0,Y 480.328,Z 820.831,A -85,B 0,C 180,E1 22960.677,E2 22960.677} C_VEL
LIN {X 0,Y 480.175,Z 828.357,A -85,B 0,C 180,E1 22958.623,E2 22958.623} C_VEL
LIN {X 0,Y 480.109,Z 834.721,A -85,B 0,C 180,E1 22956.337,E2 22956.337} C_VEL
LIN {X 0,Y 480.079,Z 838.796,A -85,B 0,C 180,E1 22954.3,E2 22954.3} C_VEL
LIN {X 0,Y 480.081,Z 841.382,A -85,B 0,C 180,E1 22952.148,E2 22952.148} C_VEL
LIN {X 0,Y 480.087,Z 842.264,A -85,B 0,C 180,E1 22950,E2 22950} C_VEL
LIN {X 0,Y 480.074,Z 841.442,A -85,B 0,C 180,E1 22947.852,E2 22947.852} C_VEL
LIN {X 0,Y 480.061,Z 838.946,A -85,B 0,C 180,E1 22945.7,E2 22945.7} C_VEL
LIN {X 0,Y 480.082,Z 834.68,A -85,B 0,C 180,E1 22943.543,E2 22943.543} C_VEL
LIN {X 0,Y 480.157,Z 828.572,A -85,B 0,C 180,E1 22941.377,E2 22941.377} C_VEL
LIN {X 0,Y 480.327,Z 820.742,A -85,B 0,C 180,E1 22939.273,E2 22939.273} C_VEL
LIN {X 0,Y 480.643,Z 811.298,A -85,B 0,C 180,E1 22937.261,E2 22937.261} C_VEL
LIN {X 0,Y 481.104,Z 800.032,A -85,B 0,C 180,E1 22935.312,E2 22935.312} C_VEL
LIN {X 0,Y 481.731,Z 787.172,A -85,B 0,C 180,E1 22933.48,E2 22933.48} C_VEL
LIN {X 0,Y 482.47,Z 773.201,A -85,B 0,C 180,E1 22931.827,E2 22931.827} C_VEL
LIN {X 0,Y 483.292,Z 758.556,A -85,B 0,C 180,E1 22930.382,E2 22930.382} C_VEL
LIN {X 0,Y 484.191,Z 742.449,A -85,B 0,C 180,E1 22929.069,E2 22929.069} C_VEL
LIN {X 0,Y 485.117,Z 724.823,A -85,B 0,C 180,E1 22927.905,E2 22927.905} C_VEL
LIN {X 0,Y 485.954,Z 707.196,A -85,B 0,C 180,E1 22926.988,E2 22926.988} C_VEL
LIN {X 0,Y 486.695,Z 688.531,A -85,B 0,C 180,E1 22926.255,E2 22926.255} C_VEL
LIN {X 0,Y 487.286,Z 669.758,A -85,B 0,C 180,E1 22925.747,E2 22925.747} C_VEL
LIN {X 0,Y 487.89,Z 616.552,A -85,B 0,C 180,E1 22924.904,E2 22924.904} C_VEL
LIN {X 0,Y 488.797,Z 545.112,A -85,B 0,C 180,E1 22923.766,E2 22923.766} C_VEL
LIN {X 0,Y 490.176,Z 478.182,A -85,B 0,C 180,E1 22922.513,E2 22922.513} C_VEL
LIN {X 0,Y 487.762,Z 457.163,A -85,B 0,C 180,E1 22921.87,E2 22921.87} C_VEL
LIN {X 0,Y 490.25,Z 412.442,A -85,B 0,C 180,E1 22918.114,E2 22918.114} C_VEL
LIN {X 0,Y 491.088,Z 396.062,A -85,B 0,C 180,E1 22916.697,E2 22916.697} C_VEL
LIN {X 0,Y 483.489,Z 374.686,A -85,B 0,C 180,E1 22914.16,E2 22914.16} C_VEL
LIN {X 0,Y 480.841,Z 366.9,A -85,B 0,C 180,E1 22913.184,E2 22913.184} C_VEL
LIN {X 0,Y 480.874,Z 366.9,A -85,B 0,C 180,E1 22909.71,E2 22909.71} C_VEL
LIN {X 0,Y 480.827,Z 366.904,A -85,B 0,C 180,E1 22906.175,E2 22906.175} C_VEL
LIN {X 0,Y 480.816,Z 366.904,A -85,B 0,C 180,E1 22902.596,E2 22902.596} C_VEL
LIN {X 0,Y 480.849,Z 366.903,A -85,B 0,C 180,E1 22899.14,E2 22899.14} C_VEL
LIN {X 0,Y 480.862,Z 366.902,A -85,B 0,C 180,E1 22895.606,E2 22895.606} C_VEL
LIN {X 0,Y 480.876,Z 366.986,A -85,B 0,C 180,E1 22893.222,E2 22893.222} C_VEL
LIN {X 0,Y 482.094,Z 370.336,A -85,B 0,C 180,E1 22892.773,E2 22892.773} C_VEL
LIN {X 0,Y 486.691,Z 382.289,A -85,B 0,C 180,E1 22891.179,E2 22891.179} C_VEL
LIN {X 0,Y 490.126,Z 394.406,A -85,B 0,C 180,E1 22889.717,E2 22889.717} C_VEL
LIN {X 0,Y 489.742,Z 411.479,A -85,B 0,C 180,E1 22888.165,E2 22888.165} C_VEL
LIN {X 0,Y 491.896,Z 424.557,A -85,B 0,C 180,E1 22887.721,E2 22887.721} C_VEL
LIN {X 0,Y 489.071,Z 536.26,A -85,B 0,C 180,E1 22885.656,E2 22885.656} C_VEL
LIN {X 0,Y 487.713,Z 619.518,A -85,B 0,C 180,E1 22884.214,E2 22884.214} C_VEL
LIN {X 0,Y 487.191,Z 638.869,A -85,B 0,C 180,E1 22883.647,E2 22883.647} C_VEL
LIN {X 0,Y 486.55,Z 656.565,A -85,B 0,C 180,E1 22882.918,E2 22882.918} C_VEL
LIN {X 0,Y 485.771,Z 673.681,A -85,B 0,C 180,E1 22882,E2 22882} C_VEL
LIN {X 0,Y 484.868,Z 690.863,A -85,B 0,C 180,E1 22880.837,E2 22880.837} C_VEL
LIN {X 0,Y 483.943,Z 706.94,A -85,B 0,C 180,E1 22879.492,E2 22879.492} C_VEL
LIN {X 0,Y 483.028,Z 721.903,A -85,B 0,C 180,E1 22877.964,E2 22877.964} C_VEL
LIN {X 0,Y 482.236,Z 734.77,A -85,B 0,C 180,E1 22876.378,E2 22876.378} C_VEL
LIN {X 0,Y 481.53,Z 746.623,A -85,B 0,C 180,E1 22874.621,E2 22874.621} C_VEL
LIN {X 0,Y 480.956,Z 757.119,A -85,B 0,C 180,E1 22872.73,E2 22872.73} C_VEL
LIN {X 0,Y 480.516,Z 766.362,A -85,B 0,C 180,E1 22870.672,E2 22870.672} C_VEL
LIN {X 0,Y 480.223,Z 773.974,A -85,B 0,C 180,E1 22868.501,E2 22868.501} C_VEL
LIN {X 0,Y 480.06,Z 779.636,A -85,B 0,C 180,E1 22866.338,E2 22866.338} C_VEL
LIN {X 0,Y 479.983,Z 783.548,A -85,B 0,C 180,E1 22864.181,E2 22864.181} C_VEL
LIN {X 0,Y 479.959,Z 785.825,A -85,B 0,C 180,E1 22862.029,E2 22862.029} C_VEL
LIN {X 0,Y 479.961,Z 786.502,A -85,B 0,C 180,E1 22859.761,E2 22859.761} C_VEL
LIN {X 0,Y 479.959,Z 785.44,A -85,B 0,C 180,E1 22857.492,E2 22857.492} C_VEL
LIN {X 0,Y 479.988,Z 782.815,A -85,B 0,C 180,E1 22855.34,E2 22855.34} C_VEL
LIN {X 0,Y 480.072,Z 778.528,A -85,B 0,C 180,E1 22853.182,E2 22853.182} C_VEL
LIN {X 0,Y 480.244,Z 772.461,A -85,B 0,C 180,E1 22851.016,E2 22851.016} C_VEL
LIN {X 0,Y 480.531,Z 764.937,A -85,B 0,C 180,E1 22848.964,E2 22848.964} C_VEL
LIN {X 0,Y 480.96,Z 756.041,A -85,B 0,C 180,E1 22847.025,E2 22847.025} C_VEL
LIN {X 0,Y 481.573,Z 745.078,A -85,B 0,C 180,E1 22845.081,E2 22845.081} C_VEL
LIN {X 0,Y 482.35,Z 732.537,A -85,B 0,C 180,E1 22843.254,E2 22843.254} C_VEL
LIN {X 0,Y 483.23,Z 718.872,A -85,B 0,C 180,E1 22841.606,E2 22841.606} C_VEL
LIN {X 0,Y 484.177,Z 704.14,A -85,B 0,C 180,E1 22840.134,E2 22840.134} C_VEL
LIN {X 0,Y 485.17,Z 687.892,A -85,B 0,C 180,E1 22838.797,E2 22838.797} C_VEL
LIN {X 0,Y 486.153,Z 670.436,A -85,B 0,C 180,E1 22837.636,E2 22837.636} C_VEL
LIN {X 0,Y 487.028,Z 652.2,A -85,B 0,C 180,E1 22836.689,E2 22836.689} C_VEL
LIN {X 0,Y 487.748,Z 633.499,A -85,B 0,C 180,E1 22835.962,E2 22835.962} C_VEL
LIN {X 0,Y 488.277,Z 614.643,A -85,B 0,C 180,E1 22835.453,E2 22835.453} C_VEL
LIN {X 0,Y 491.256,Z 422.615,A -85,B 0,C 180,E1 22832.262,E2 22832.262} C_VEL
LIN {X 0,Y 488.294,Z 406.516,A -85,B 0,C 180,E1 22831.77,E2 22831.77} C_VEL
LIN {X 0,Y 488.765,Z 392.246,A -85,B 0,C 180,E1 22830.391,E2 22830.391} C_VEL
LIN {X 0,Y 483.183,Z 374.157,A -85,B 0,C 180,E1 22828.216,E2 22828.216} C_VEL
LIN {X 0,Y 481.099,Z 371.22,A -85,B 0,C 180,E1 22827.743,E2 22827.743} C_VEL
LIN {X 0,Y 476.895,Z 368.873,A -85,B 0,C 180,E1 22827.013,E2 22827.013} C_VEL
LIN {X 0,Y 473.716,Z 368.027,A -85,B 0,C 180,E1 22826.273,E2 22826.273} C_VEL
LIN {X 0,Y 472.884,Z 367.893,A -85,B 0,C 180,E1 22825.728,E2 22825.728} C_VEL
LIN {X 0,Y 472.913,Z 367.889,A -85,B 0,C 180,E1 22822.183,E2 22822.183} C_VEL
LIN {X 0,Y 472.924,Z 367.891,A -85,B 0,C 180,E1 22818.728,E2 22818.728} C_VEL
LIN {X 0,Y 472.884,Z 367.891,A -85,B 0,C 180,E1 22815.244,E2 22815.244} C_VEL
LIN {X 0,Y 472.883,Z 367.889,A -85,B 0,C 180,E1 22811.54,E2 22811.54} C_VEL
LIN {X 0,Y 472.923,Z 367.89,A -85,B 0,C 180,E1 22808.123,E2 22808.123} C_VEL
LIN {X 0,Y 472.911,Z 367.891,A -85,B 0,C 180,E1 22804.662,E2 22804.662} C_VEL
LIN {X 0,Y 472.882,Z 367.89,A -85,B 0,C 180,E1 22801.2,E2 22801.2} C_VEL
LIN {X 0,Y 472.889,Z 367.889,A -85,B 0,C 180,E1 22797.584,E2 22797.584} C_VEL
LIN {X 0,Y 472.929,Z 367.888,A -85,B 0,C 180,E1 22794.03,E2 22794.03} C_VEL
LIN {X 0,Y 472.915,Z 367.887,A -85,B 0,C 180,E1 22790.509,E2 22790.509} C_VEL
LIN {X 0,Y 472.883,Z 367.887,A -85,B 0,C 180,E1 22786.965,E2 22786.965} C_VEL
LIN {X 0,Y 472.882,Z 367.887,A -85,B 0,C 180,E1 22783.325,E2 22783.325} C_VEL
LIN {X 0,Y 472.924,Z 367.888,A -85,B 0,C 180,E1 22779.861,E2 22779.861} C_VEL
LIN {X 0,Y 472.905,Z 367.889,A -85,B 0,C 180,E1 22776.423,E2 22776.423} C_VEL
LIN {X 0,Y 472.878,Z 367.887,A -85,B 0,C 180,E1 22772.909,E2 22772.909} C_VEL
LIN {X 0,Y 472.886,Z 367.887,A -85,B 0,C 180,E1 22769.273,E2 22769.273} C_VEL
LIN {X 0,Y 472.925,Z 367.89,A -85,B 0,C 180,E1 22765.756,E2 22765.756} C_VEL
LIN {X 0,Y 472.908,Z 367.886,A -85,B 0,C 180,E1 22762.223,E2 22762.223} C_VEL
LIN {X 0,Y 472.878,Z 367.889,A -85,B 0,C 180,E1 22758.783,E2 22758.783} C_VEL
LIN {X 0,Y 472.888,Z 367.891,A -85,B 0,C 180,E1 22755.177,E2 22755.177} C_VEL
LIN {X 0,Y 472.93,Z 367.892,A -85,B 0,C 180,E1 22751.638,E2 22751.638} C_VEL
LIN {X 0,Y 472.913,Z 367.889,A -85,B 0,C 180,E1 22748.024,E2 22748.024} C_VEL
LIN {X 0,Y 472.88,Z 367.889,A -85,B 0,C 180,E1 22744.536,E2 22744.536} C_VEL
LIN {X 0,Y 472.881,Z 367.889,A -85,B 0,C 180,E1 22740.839,E2 22740.839} C_VEL
LIN {X 0,Y 472.918,Z 367.893,A -85,B 0,C 180,E1 22737.375,E2 22737.375} C_VEL
LIN {X 0,Y 472.914,Z 367.892,A -85,B 0,C 180,E1 22733.851,E2 22733.851} C_VEL
LIN {X 0,Y 472.877,Z 367.892,A -85,B 0,C 180,E1 22730.473,E2 22730.473} C_VEL
LIN {X 0,Y 472.89,Z 367.891,A -85,B 0,C 180,E1 22726.926,E2 22726.926} C_VEL
LIN {X 0,Y 472.931,Z 367.891,A -85,B 0,C 180,E1 22723.402,E2 22723.402} C_VEL
LIN {X 0,Y 472.899,Z 367.892,A -85,B 0,C 180,E1 22719.87,E2 22719.87} C_VEL
LIN {X 0,Y 472.876,Z 367.893,A -85,B 0,C 180,E1 22716.332,E2 22716.332} C_VEL
LIN {X 0,Y 472.886,Z 367.895,A -85,B 0,C 180,E1 22712.698,E2 22712.698} C_VEL
LIN {X 0,Y 472.908,Z 368.119,A -85,B 0,C 180,E1 22712.195,E2 22712.195} C_VEL
LIN {X 0,Y 478.256,Z 388.002,A -85,B 0,C 180,E1 22709.086,E2 22709.086} C_VEL
LIN {X 0,Y 478.974,Z 391.993,A -85,B 0,C 180,E1 22708.497,E2 22708.497} C_VEL
LIN {X 0,Y 477.488,Z 419.66,A -85,B 0,C 180,E1 22704.891,E2 22704.891} C_VEL
LIN {X 0,Y 476.119,Z 448.566,A -85,B 0,C 180,E1 22701.174,E2 22701.174} C_VEL
LIN {X 0,Y 474.956,Z 477.449,A -85,B 0,C 180,E1 22697.514,E2 22697.514} C_VEL
LIN {X 0,Y 474.924,Z 479.924,A -85,B 0,C 180,E1 22697.235,E2 22697.235} C_VEL
LIN {X 0,Y 477.196,Z 496.322,A -85,B 0,C 180,E1 22696.833,E2 22696.833} C_VEL
LIN {X 0,Y 475.715,Z 598.28,A -85,B 0,C 180,E1 22695.025,E2 22695.025} C_VEL
LIN {X 0,Y 475.463,Z 613.02,A -85,B 0,C 180,E1 22694.555,E2 22694.555} C_VEL
LIN {X 0,Y 475.073,Z 628.599,A -85,B 0,C 180,E1 22693.81,E2 22693.81} C_VEL
LIN {X 0,Y 474.557,Z 643.214,A -85,B 0,C 180,E1 22692.843,E2 22692.843} C_VEL
LIN {X 0,Y 474.11,Z 655.281,A -85,B 0,C 180,E1 22691.804,E2 22691.804} C_VEL
LIN {X 0,Y 473.696,Z 666.59,A -85,B 0,C 180,E1 22690.582,E2 22690.582} C_VEL
LIN {X 0,Y 473.281,Z 677.203,A -85,B 0,C 180,E1 22689.117,E2 22689.117} C_VEL
LIN {X 0,Y 472.99,Z 685.517,A -85,B 0,C 180,E1 22687.653,E2 22687.653} C_VEL
LIN {X 0,Y 472.772,Z 692.496,A -85,B 0,C 180,E1 22686.07,E2 22686.07} C_VEL
LIN {X 0,Y 472.633,Z 697.951,A -85,B 0,C 180,E1 22684.368,E2 22684.368} C_VEL
LIN {X 0,Y 472.574,Z 701.657,A -85,B 0,C 180,E1 22682.668,E2 22682.668} C_VEL
LIN {X 0,Y 472.575,Z 703.817,A -85,B 0,C 180,E1 22680.728,E2 22680.728} C_VEL
LIN {X 0,Y 472.603,Z 703.911,A -85,B 0,C 180,E1 22678.909,E2 22678.909} C_VEL
LIN {X 0,Y 472.687,Z 702.373,A -85,B 0,C 180,E1 22677.212,E2 22677.212} C_VEL
LIN {X 0,Y 472.832,Z 698.819,A -85,B 0,C 180,E1 22675.391,E2 22675.391} C_VEL
LIN {X 0,Y 473.048,Z 693.614,A -85,B 0,C 180,E1 22673.69,E2 22673.69} C_VEL
LIN {X 0,Y 473.344,Z 686.969,A -85,B 0,C 180,E1 22672.108,E2 22672.108} C_VEL
LIN {X 0,Y 473.733,Z 678.12,A -85,B 0,C 180,E1 22670.525,E2 22670.525} C_VEL
LIN {X 0,Y 474.197,Z 668.015,A -85,B 0,C 180,E1 22669.122,E2 22669.122} C_VEL
LIN {X 0,Y 474.689,Z 656.911,A -85,B 0,C 180,E1 22667.902,E2 22667.902} C_VEL
LIN {X 0,Y 475.224,Z 643.321,A -85,B 0,C 180,E1 22666.742,E2 22666.742} C_VEL
LIN {X 0,Y 475.742,Z 629.201,A -85,B 0,C 180,E1 22665.827,E2 22665.827} C_VEL
LIN {X 0,Y 476.158,Z 614.632,A -85,B 0,C 180,E1 22665.125,E2 22665.125} C_VEL
LIN {X 0,Y 476.491,Z 598.813,A -85,B 0,C 180,E1 22664.607,E2 22664.607} C_VEL
LIN {X 0,Y 479.356,Z 495.573,A -85,B 0,C 180,E1 22662.368,E2 22662.368} C_VEL
LIN {X 0,Y 476.473,Z 479.741,A -85,B 0,C 180,E1 22661.78,E2 22661.78} C_VEL
LIN {X 0,Y 478.252,Z 450.384,A -85,B 0,C 180,E1 22657.894,E2 22657.894} C_VEL
LIN {X 0,Y 480.408,Z 422.57,A -85,B 0,C 180,E1 22654.083,E2 22654.083} C_VEL
LIN {X 0,Y 482.8,Z 398.366,A -85,B 0,C 180,E1 22650.641,E2 22650.641} C_VEL
LIN {X 0,Y 480.118,Z 388.049,A -85,B 0,C 180,E1 22648.625,E2 22648.625} C_VEL
LIN {X 0,Y 477.141,Z 378.662,A -85,B 0,C 180,E1 22646.514,E2 22646.514} C_VEL
LIN {X 0,Y 474.167,Z 371.272,A -85,B 0,C 180,E1 22644.484,E2 22644.484} C_VEL
LIN {X 0,Y 472.879,Z 367.897,A -85,B 0,C 180,E1 22643.397,E2 22643.397} C_VEL
LIN {X 0,Y 472.88,Z 367.895,A -85,B 0,C 180,E1 22639.684,E2 22639.684} C_VEL
LIN {X 0,Y 472.922,Z 367.891,A -85,B 0,C 180,E1 22636.263,E2 22636.263} C_VEL
LIN {X 0,Y 472.925,Z 367.891,A -85,B 0,C 180,E1 22632.63,E2 22632.63} C_VEL
LIN {X 0,Y 472.949,Z 368.101,A -85,B 0,C 180,E1 22630.151,E2 22630.151} C_VEL
LIN {X 0,Y 474.265,Z 371.491,A -85,B 0,C 180,E1 22629.233,E2 22629.233} C_VEL
LIN {X 0,Y 475.123,Z 373.176,A -85,B 0,C 180,E1 22628.778,E2 22628.778} C_VEL
LIN {X 0,Y 478.237,Z 380.252,A -85,B 0,C 180,E1 22627.173,E2 22627.173} C_VEL
LIN {X 0,Y 482.346,Z 391.225,A -85,B 0,C 180,E1 22625.189,E2 22625.189} C_VEL
LIN {X 0,Y 485.282,Z 401.093,A -85,B 0,C 180,E1 22623.73,E2 22623.73} C_VEL
LIN {X 0,Y 481.83,Z 435.913,A -85,B 0,C 180,E1 22620.42,E2 22620.42} C_VEL
LIN {X 0,Y 480.318,Z 458.586,A -85,B 0,C 180,E1 22618.427,E2 22618.427} C_VEL
LIN {X 0,Y 483.122,Z 482.22,A -85,B 0,C 180,E1 22617.814,E2 22617.814} C_VEL
LIN {X 0,Y 479.927,Z 670.781,A -85,B 0,C 180,E1 22614.604,E2 22614.604} C_VEL
LIN {X 0,Y 479.259,Z 689.569,A -85,B 0,C 180,E1 22614.071,E2 22614.071} C_VEL
LIN {X 0,Y 478.44,Z 708.133,A -85,B 0,C 180,E1 22613.315,E2 22613.315} C_VEL
LIN {X 0,Y 477.494,Z 726.263,A -85,B 0,C 180,E1 22612.337,E2 22612.337} C_VEL
LIN {X 0,Y 476.501,Z 743.54,A -85,B 0,C 180,E1 22611.156,E2 22611.156} C_VEL
LIN {X 0,Y 475.513,Z 759.776,A -85,B 0,C 180,E1 22609.788,E2 22609.788} C_VEL
LIN {X 0,Y 474.595,Z 774.958,A -85,B 0,C 180,E1 22608.231,E2 22608.231} C_VEL
LIN {X 0,Y 473.801,Z 788.54,A -85,B 0,C 180,E1 22606.552,E2 22606.552} C_VEL
LIN {X 0,Y 473.137,Z 801.029,A -85,B 0,C 180,E1 22604.69,E2 22604.69} C_VEL
LIN {X 0,Y 472.654,Z 811.923,A -85,B 0,C 180,E1 22602.709,E2 22602.709} C_VEL
LIN {X 0,Y 472.336,Z 820.771,A -85,B 0,C 180,E1 22600.736,E2 22600.736} C_VEL
LIN {X 0,Y 472.175,Z 828.218,A -85,B 0,C 180,E1 22598.647,E2 22598.647} C_VEL
LIN {X 0,Y 472.111,Z 833.891,A -85,B 0,C 180,E1 22596.567,E2 22596.567} C_VEL
LIN {X 0,Y 472.099,Z 838.096,A -85,B 0,C 180,E1 22594.373,E2 22594.373} C_VEL
LIN {X 0,Y 472.118,Z 840.572,A -85,B 0,C 180,E1 22592.185,E2 22592.185} C_VEL
LIN {X 0,Y 472.137,Z 841.37,A -85,B 0,C 180,E1 22590,E2 22590} C_VEL
LIN {X 0,Y 472.125,Z 840.492,A -85,B 0,C 180,E1 22587.815,E2 22587.815} C_VEL
LIN {X 0,Y 472.109,Z 837.932,A -85,B 0,C 180,E1 22585.627,E2 22585.627} C_VEL
LIN {X 0,Y 472.118,Z 833.639,A -85,B 0,C 180,E1 22583.433,E2 22583.433} C_VEL
LIN {X 0,Y 472.181,Z 827.836,A -85,B 0,C 180,E1 22581.353,E2 22581.353} C_VEL
LIN {X 0,Y 472.354,Z 819.754,A -85,B 0,C 180,E1 22579.141,E2 22579.141} C_VEL
LIN {X 0,Y 472.689,Z 810.044,A -85,B 0,C 180,E1 22577.043,E2 22577.043} C_VEL
LIN {X 0,Y 473.17,Z 798.712,A -85,B 0,C 180,E1 22575.06,E2 22575.06} C_VEL
LIN {X 0,Y 473.792,Z 786.737,A -85,B 0,C 180,E1 22573.321,E2 22573.321} C_VEL
LIN {X 0,Y 474.57,Z 772.854,A -85,B 0,C 180,E1 22571.64,E2 22571.64} C_VEL
LIN {X 0,Y 475.441,Z 758.237,A -85,B 0,C 180,E1 22570.166,E2 22570.166} C_VEL
LIN {X 0,Y 476.389,Z 742.328,A -85,B 0,C 180,E1 22568.838,E2 22568.838} C_VEL
LIN {X 0,Y 477.374,Z 724.862,A -85,B 0,C 180,E1 22567.657,E2 22567.657} C_VEL
LIN {X 0,Y 478.285,Z 707.017,A -85,B 0,C 180,E1 22566.707,E2 22566.707} C_VEL
LIN {X 0,Y 479.08,Z 688.292,A -85,B 0,C 180,E1 22565.956,E2 22565.956} C_VEL
LIN {X 0,Y 479.714,Z 669.417,A -85,B 0,C 180,E1 22565.434,E2 22565.434} C_VEL
LIN {X 0,Y 480.293,Z 623.287,A -85,B 0,C 180,E1 22564.686,E2 22564.686} C_VEL
LIN {X 0,Y 481.027,Z 572.063,A -85,B 0,C 180,E1 22563.841,E2 22563.841} C_VEL
LIN {X 0,Y 483.226,Z 479.351,A -85,B 0,C 180,E1 22562.062,E2 22562.062} C_VEL
LIN {X 0,Y 480.45,Z 454.744,A -85,B 0,C 180,E1 22561.267,E2 22561.267} C_VEL
LIN {X 0,Y 483.073,Z 411.694,A -85,B 0,C 180,E1 22557.583,E2 22557.583} C_VEL
LIN {X 0,Y 483.833,Z 398.941,A -85,B 0,C 180,E1 22556.46,E2 22556.46} C_VEL
LIN {X 0,Y 475.972,Z 376.639,A -85,B 0,C 180,E1 22553.77,E2 22553.77} C_VEL
LIN {X 0,Y 472.88,Z 367.893,A -85,B 0,C 180,E1 22552.639,E2 22552.639} C_VEL
LIN {X 0,Y 472.908,Z 367.891,A -85,B 0,C 180,E1 22549.193,E2 22549.193} C_VEL
LIN {X 0,Y 472.933,Z 367.889,A -85,B 0,C 180,E1 22545.59,E2 22545.59} C_VEL
LIN {X 0,Y 472.89,Z 367.894,A -85,B 0,C 180,E1 22542.086,E2 22542.086} C_VEL
LIN {X 0,Y 472.878,Z 367.895,A -85,B 0,C 180,E1 22538.525,E2 22538.525} C_VEL
LIN {X 0,Y 472.898,Z 367.894,A -85,B 0,C 180,E1 22534.958,E2 22534.958} C_VEL
LIN {X 0,Y 472.904,Z 368.015,A -85,B 0,C 180,E1 22534.023,E2 22534.023} C_VEL
LIN {X 0,Y 474.228,Z 371.366,A -85,B 0,C 180,E1 22533.532,E2 22533.532} C_VEL
LIN {X 0,Y 479.247,Z 383.756,A -85,B 0,C 180,E1 22531.769,E2 22531.769} C_VEL
LIN {X 0,Y 483.157,Z 396.895,A -85,B 0,C 180,E1 22530.114,E2 22530.114} C_VEL
LIN {X 0,Y 482.892,Z 412.361,A -85,B 0,C 180,E1 22528.691,E2 22528.691} C_VEL
LIN {X 0,Y 485.077,Z 425.739,A -85,B 0,C 180,E1 22528.199,E2 22528.199} C_VEL
LIN {X 0,Y 482.014,Z 530.873,A -85,B 0,C 180,E1 22526.173,E2 22526.173} C_VEL
LIN {X 0,Y 480.3,Z 620.609,A -85,B 0,C 180,E1 22524.554,E2 22524.554} C_VEL
LIN {X 0,Y 479.73,Z 639.883,A -85,B 0,C 180,E1 22523.971,E2 22523.971} C_VEL
LIN {X 0,Y 478.986,Z 658.618,A -85,B 0,C 180,E1 22523.171,E2 22523.171} C_VEL
LIN {X 0,Y 478.11,Z 676.373,A -85,B 0,C 180,E1 22522.177,E2 22522.177} C_VEL
LIN {X 0,Y 477.16,Z 693.134,A -85,B 0,C 180,E1 22520.997,E2 22520.997} C_VEL
LIN {X 0,Y 476.181,Z 708.896,A -85,B 0,C 180,E1 22519.631,E2 22519.631} C_VEL
LIN {X 0,Y 475.218,Z 723.62,A -85,B 0,C 180,E1 22518.08,E2 22518.08} C_VEL
LIN {X 0,Y 474.35,Z 736.75,A -85,B 0,C 180,E1 22516.406,E2 22516.406} C_VEL
LIN {X 0,Y 473.588,Z 748.782,A -85,B 0,C 180,E1 22514.551,E2 22514.551} C_VEL
LIN {X 0,Y 472.98,Z 759.222,A -85,B 0,C 180,E1 22512.576,E2 22512.576} C_VEL
LIN {X 0,Y 472.552,Z 767.663,A -85,B 0,C 180,E1 22510.607,E2 22510.607} C_VEL
LIN {X 0,Y 472.259,Z 774.731,A -85,B 0,C 180,E1 22508.523,E2 22508.523} C_VEL
LIN {X 0,Y 472.084,Z 780.327,A -85,B 0,C 180,E1 22506.323,E2 22506.323} C_VEL
LIN {X 0,Y 472,Z 784.164,A -85,B 0,C 180,E1 22504.13,E2 22504.13} C_VEL
LIN {X 0,Y 471.972,Z 786.357,A -85,B 0,C 180,E1 22501.942,E2 22501.942} C_VEL
LIN {X 0,Y 471.974,Z 786.963,A -85,B 0,C 180,E1 22499.757,E2 22499.757} C_VEL
LIN {X 0,Y 471.972,Z 785.995,A -85,B 0,C 180,E1 22497.572,E2 22497.572} C_VEL
LIN {X 0,Y 472.004,Z 783.432,A -85,B 0,C 180,E1 22495.383,E2 22495.383} C_VEL
LIN {X 0,Y 472.095,Z 779.203,A -85,B 0,C 180,E1 22493.188,E2 22493.188} C_VEL
LIN {X 0,Y 472.28,Z 773.19,A -85,B 0,C 180,E1 22490.986,E2 22490.986} C_VEL
LIN {X 0,Y 472.588,Z 765.723,A -85,B 0,C 180,E1 22488.899,E2 22488.899} C_VEL
LIN {X 0,Y 473.046,Z 756.889,A -85,B 0,C 180,E1 22486.929,E2 22486.929} C_VEL
LIN {X 0,Y 473.698,Z 745.991,A -85,B 0,C 180,E1 22484.952,E2 22484.952} C_VEL
LIN {X 0,Y 474.523,Z 733.525,A -85,B 0,C 180,E1 22483.095,E2 22483.095} C_VEL
LIN {X 0,Y 475.492,Z 719.401,A -85,B 0,C 180,E1 22481.36,E2 22481.36} C_VEL
LIN {X 0,Y 476.499,Z 704.759,A -85,B 0,C 180,E1 22479.871,E2 22479.871} C_VEL
LIN {X 0,Y 477.505,Z 689.257,A -85,B 0,C 180,E1 22478.568,E2 22478.568} C_VEL
LIN {X 0,Y 478.463,Z 673.251,A -85,B 0,C 180,E1 22477.468,E2 22477.468} C_VEL
LIN {X 0,Y 479.38,Z 656.08,A -85,B 0,C 180,E1 22476.523,E2 22476.523} C_VEL
LIN {X 0,Y 480.175,Z 637.632,A -85,B 0,C 180,E1 22475.745,E2 22475.745} C_VEL
LIN {X 0,Y 480.794,Z 618.357,A -85,B 0,C 180,E1 22475.169,E2 22475.169} C_VEL
LIN {X 0,Y 481.316,Z 587.13,A -85,B 0,C 180,E1 22474.613,E2 22474.613} C_VEL
LIN {X 0,Y 484.134,Z 423.953,A -85,B 0,C 180,E1 22471.853,E2 22471.853} C_VEL
LIN {X 0,Y 481.02,Z 406.719,A -85,B 0,C 180,E1 22471.304,E2 22471.304} C_VEL
LIN {X 0,Y 481.49,Z 395.137,A -85,B 0,C 180,E1 22470.182,E2 22470.182} C_VEL
LIN {X 0,Y 475.598,Z 376.099,A -85,B 0,C 180,E1 22467.867,E2 22467.867} C_VEL
LIN {X 0,Y 472.924,Z 367.892,A -85,B 0,C 180,E1 22466.829,E2 22466.829} C_VEL
LIN {X 0,Y 472.884,Z 367.893,A -85,B 0,C 180,E1 22465.728,E2 22465.728} C_VEL
LIN {X 0,Y 471.882,Z 368.02,A -85,B 0,C 180,E1 22464.795,E2 22464.795} C_VEL
LIN {X 0,Y 465.377,Z 368.829,A -85,B 0,C 180,E1 22462.101,E2 22462.101} C_VEL
LIN {X 0,Y 464.945,Z 368.881,A -85,B 0,C 180,E1 22461.484,E2 22461.484} C_VEL
LIN {X 0,Y 464.954,Z 368.88,A -85,B 0,C 180,E1 22457.86,E2 22457.86} C_VEL
LIN {X 0,Y 464.991,Z 368.879,A -85,B 0,C 180,E1 22454.271,E2 22454.271} C_VEL
LIN {X 0,Y 464.988,Z 368.877,A -85,B 0,C 180,E1 22450.619,E2 22450.619} C_VEL
LIN {X 0,Y 464.946,Z 368.879,A -85,B 0,C 180,E1 22447.178,E2 22447.178} C_VEL
LIN {X 0,Y 464.943,Z 368.88,A -85,B 0,C 180,E1 22443.447,E2 22443.447} C_VEL
LIN {X 0,Y 464.972,Z 368.878,A -85,B 0,C 180,E1 22439.926,E2 22439.926} C_VEL
LIN {X 0,Y 464.987,Z 368.877,A -85,B 0,C 180,E1 22436.431,E2 22436.431} C_VEL
LIN {X 0,Y 464.948,Z 368.877,A -85,B 0,C 180,E1 22432.907,E2 22432.907} C_VEL
LIN {X 0,Y 464.942,Z 368.879,A -85,B 0,C 180,E1 22429.252,E2 22429.252} C_VEL
LIN {X 0,Y 464.965,Z 368.88,A -85,B 0,C 180,E1 22425.721,E2 22425.721} C_VEL
LIN {X 0,Y 464.994,Z 368.876,A -85,B 0,C 180,E1 22422.165,E2 22422.165} C_VEL
LIN {X 0,Y 464.96,Z 368.875,A -85,B 0,C 180,E1 22418.533,E2 22418.533} C_VEL
LIN {X 0,Y 464.94,Z 368.877,A -85,B 0,C 180,E1 22415.058,E2 22415.058} C_VEL
LIN {X 0,Y 464.957,Z 368.879,A -85,B 0,C 180,E1 22411.479,E2 22411.479} C_VEL
LIN {X 0,Y 464.993,Z 368.874,A -85,B 0,C 180,E1 22408.028,E2 22408.028} C_VEL
LIN {X 0,Y 464.954,Z 368.878,A -85,B 0,C 180,E1 22404.447,E2 22404.447} C_VEL
LIN {X 0,Y 464.94,Z 368.878,A -85,B 0,C 180,E1 22400.968,E2 22400.968} C_VEL
LIN {X 0,Y 464.967,Z 368.878,A -85,B 0,C 180,E1 22397.456,E2 22397.456} C_VEL
LIN {X 0,Y 464.985,Z 368.879,A -85,B 0,C 180,E1 22393.985,E2 22393.985} C_VEL
LIN {X 0,Y 464.948,Z 368.88,A -85,B 0,C 180,E1 22390.398,E2 22390.398} C_VEL
LIN {X 0,Y 464.941,Z 368.878,A -85,B 0,C 180,E1 22386.825,E2 22386.825} C_VEL
LIN {X 0,Y 464.967,Z 368.878,A -85,B 0,C 180,E1 22383.293,E2 22383.293} C_VEL
LIN {X 0,Y 465.007,Z 368.877,A -85,B 0,C 180,E1 22379.649,E2 22379.649} C_VEL
LIN {X 0,Y 464.963,Z 368.881,A -85,B 0,C 180,E1 22376.006,E2 22376.006} C_VEL
LIN {X 0,Y 464.938,Z 368.882,A -85,B 0,C 180,E1 22372.511,E2 22372.511} C_VEL
LIN {X 0,Y 464.956,Z 368.879,A -85,B 0,C 180,E1 22369.009,E2 22369.009} C_VEL
LIN {X 0,Y 464.991,Z 368.879,A -85,B 0,C 180,E1 22365.493,E2 22365.493} C_VEL
LIN {X 0,Y 464.957,Z 368.881,A -85,B 0,C 180,E1 22361.922,E2 22361.922} C_VEL
LIN {X 0,Y 464.936,Z 368.882,A -85,B 0,C 180,E1 22358.426,E2 22358.426} C_VEL
LIN {X 0,Y 464.957,Z 368.883,A -85,B 0,C 180,E1 22354.891,E2 22354.891} C_VEL
LIN {X 0,Y 464.964,Z 369.029,A -85,B 0,C 180,E1 22352.643,E2 22352.643} C_VEL
LIN {X 0,Y 470.448,Z 389.386,A -85,B 0,C 180,E1 22349.403,E2 22349.403} C_VEL
LIN {X 0,Y 471.421,Z 393.967,A -85,B 0,C 180,E1 22348.711,E2 22348.711} C_VEL
LIN {X 0,Y 469.835,Z 421.631,A -85,B 0,C 180,E1 22345.056,E2 22345.056} C_VEL
LIN {X 0,Y 468.399,Z 450.166,A -85,B 0,C 180,E1 22341.343,E2 22341.343} C_VEL
LIN {X 0,Y 467.145,Z 479.316,A -85,B 0,C 180,E1 22337.598,E2 22337.598} C_VEL
LIN {X 0,Y 469.611,Z 497.239,A -85,B 0,C 180,E1 22337.131,E2 22337.131} C_VEL
LIN {X 0,Y 468.008,Z 598.819,A -85,B 0,C 180,E1 22335.279,E2 22335.279} C_VEL
LIN {X 0,Y 467.722,Z 614.285,A -85,B 0,C 180,E1 22334.769,E2 22334.769} C_VEL
LIN {X 0,Y 467.334,Z 628.932,A -85,B 0,C 180,E1 22334.056,E2 22334.056} C_VEL
LIN {X 0,Y 466.813,Z 643.013,A -85,B 0,C 180,E1 22333.123,E2 22333.123} C_VEL
LIN {X 0,Y 466.333,Z 655.357,A -85,B 0,C 180,E1 22332.067,E2 22332.067} C_VEL
LIN {X 0,Y 465.867,Z 667.365,A -85,B 0,C 180,E1 22330.762,E2 22330.762} C_VEL
LIN {X 0,Y 465.423,Z 678.061,A -85,B 0,C 180,E1 22329.272,E2 22329.272} C_VEL
LIN {X 0,Y 465.111,Z 686.445,A -85,B 0,C 180,E1 22327.784,E2 22327.784} C_VEL
LIN {X 0,Y 464.876,Z 693.492,A -85,B 0,C 180,E1 22326.174,E2 22326.174} C_VEL
LIN {X 0,Y 464.726,Z 699.022,A -85,B 0,C 180,E1 22324.442,E2 22324.442} C_VEL
LIN {X 0,Y 464.661,Z 702.777,A -85,B 0,C 180,E1 22322.714,E2 22322.714} C_VEL
LIN {X 0,Y 464.662,Z 704.99,A -85,B 0,C 180,E1 22320.74,E2 22320.74} C_VEL
LIN {X 0,Y 464.697,Z 705.128,A -85,B 0,C 180,E1 22318.891,E2 22318.891} C_VEL
LIN {X 0,Y 464.795,Z 703.626,A -85,B 0,C 180,E1 22317.164,E2 22317.164} C_VEL
LIN {X 0,Y 464.961,Z 700.107,A -85,B 0,C 180,E1 22315.313,E2 22315.313} C_VEL
LIN {X 0,Y 465.205,Z 694.932,A -85,B 0,C 180,E1 22313.583,E2 22313.583} C_VEL
LIN {X 0,Y 465.539,Z 688.118,A -85,B 0,C 180,E1 22311.938,E2 22311.938} C_VEL
LIN {X 0,Y 465.954,Z 679.451,A -85,B 0,C 180,E1 22310.365,E2 22310.365} C_VEL
LIN {X 0,Y 466.455,Z 669.367,A -85,B 0,C 180,E1 22308.94,E2 22308.94} C_VEL
LIN {X 0,Y 467.018,Z 657.723,A -85,B 0,C 180,E1 22307.638,E2 22307.638} C_VEL
LIN {X 0,Y 467.609,Z 644.132,A -85,B 0,C 180,E1 22306.459,E2 22306.459} C_VEL
LIN {X 0,Y 468.209,Z 628.94,A -85,B 0,C 180,E1 22305.468,E2 22305.468} C_VEL
LIN {X 0,Y 468.653,Z 613.876,A -85,B 0,C 180,E1 22304.755,E2 22304.755} C_VEL
LIN {X 0,Y 468.986,Z 598.426,A -85,B 0,C 180,E1 22304.259,E2 22304.259} C_VEL
LIN {X 0,Y 472.281,Z 498.062,A -85,B 0,C 180,E1 22301.988,E2 22301.988} C_VEL
LIN {X 0,Y 469.086,Z 479.511,A -85,B 0,C 180,E1 22301.257,E2 22301.257} C_VEL
LIN {X 0,Y 471.1,Z 450.059,A -85,B 0,C 180,E1 22297.277,E2 22297.277} C_VEL
LIN {X 0,Y 473.421,Z 423.406,A -85,B 0,C 180,E1 22293.537,E2 22293.537} C_VEL
LIN {X 0,Y 475.766,Z 401.499,A -85,B 0,C 180,E1 22290.336,E2 22290.336} C_VEL
LIN {X 0,Y 473.105,Z 390.865,A -85,B 0,C 180,E1 22288.167,E2 22288.167} C_VEL
LIN {X 0,Y 470.111,Z 381.919,A -85,B 0,C 180,E1 22285.988,E2 22285.988} C_VEL
LIN {X 0,Y 467.888,Z 376.121,A -85,B 0,C 180,E1 22284.297,E2 22284.297} C_VEL
LIN {X 0,Y 466.436,Z 372.618,A -85,B 0,C 180,E1 22283.089,E2 22283.089} C_VEL
LIN {X 0,Y 464.94,Z 368.886,A -85,B 0,C 180,E1 22281.517,E2 22281.517} C_VEL
LIN {X 0,Y 464.961,Z 368.883,A -85,B 0,C 180,E1 22278.027,E2 22278.027} C_VEL
LIN {X 0,Y 464.995,Z 368.878,A -85,B 0,C 180,E1 22274.448,E2 22274.448} C_VEL
LIN {X 0,Y 464.985,Z 369.003,A -85,B 0,C 180,E1 22272.03,E2 22272.03} C_VEL
LIN {X 0,Y 466.51,Z 372.676,A -85,B 0,C 180,E1 22270.659,E2 22270.659} C_VEL
LIN {X 0,Y 467.245,Z 374.037,A -85,B 0,C 180,E1 22270.187,E2 22270.187} C_VEL
LIN {X 0,Y 469.455,Z 379.121,A -85,B 0,C 180,E1 22268.768,E2 22268.768} C_VEL
LIN {X 0,Y 472.254,Z 385.714,A -85,B 0,C 180,E1 22267.244,E2 22267.244} C_VEL
LIN {X 0,Y 475.89,Z 395.636,A -85,B 0,C 180,E1 22265.393,E2 22265.393} C_VEL
LIN {X 0,Y 478.39,Z 404.246,A -85,B 0,C 180,E1 22264.065,E2 22264.065} C_VEL
LIN {X 0,Y 474.798,Z 436.303,A -85,B 0,C 180,E1 22260.92,E2 22260.92} C_VEL
LIN {X 0,Y 473.075,Z 458.758,A -85,B 0,C 180,E1 22258.885,E2 22258.885} C_VEL
LIN {X 0,Y 475.978,Z 483.126,A -85,B 0,C 180,E1 22258.235,E2 22258.235} C_VEL
LIN {X 0,Y 472.502,Z 670.358,A -85,B 0,C 180,E1 22254.971,E2 22254.971} C_VEL
LIN {X 0,Y 471.787,Z 689.174,A -85,B 0,C 180,E1 22254.428,E2 22254.428} C_VEL
LIN {X 0,Y 470.909,Z 707.772,A -85,B 0,C 180,E1 22253.659,E2 22253.659} C_VEL
LIN {X 0,Y 469.938,Z 725.108,A -85,B 0,C 180,E1 22252.716,E2 22252.716} C_VEL
LIN {X 0,Y 468.862,Z 742.537,A -85,B 0,C 180,E1 22251.518,E2 22251.518} C_VEL
LIN {X 0,Y 467.796,Z 758.896,A -85,B 0,C 180,E1 22250.128,E2 22250.128} C_VEL
LIN {X 0,Y 466.836,Z 773.598,A -85,B 0,C 180,E1 22248.61,E2 22248.61} C_VEL
LIN {X 0,Y 466.001,Z 786.869,A -85,B 0,C 180,E1 22246.966,E2 22246.966} C_VEL
LIN {X 0,Y 465.3,Z 798.8,A -85,B 0,C 180,E1 22245.198,E2 22245.198} C_VEL
LIN {X 0,Y 464.792,Z 809.415,A -85,B 0,C 180,E1 22243.308,E2 22243.308} C_VEL
LIN {X 0,Y 464.414,Z 818.67,A -85,B 0,C 180,E1 22241.298,E2 22241.298} C_VEL
LIN {X 0,Y 464.212,Z 826.5,A -85,B 0,C 180,E1 22239.171,E2 22239.171} C_VEL
LIN {X 0,Y 464.137,Z 832.494,A -85,B 0,C 180,E1 22237.053,E2 22237.053} C_VEL
LIN {X 0,Y 464.11,Z 837.023,A -85,B 0,C 180,E1 22234.82,E2 22234.82} C_VEL
LIN {X 0,Y 464.124,Z 839.788,A -85,B 0,C 180,E1 22232.593,E2 22232.593} C_VEL
LIN {X 0,Y 464.143,Z 840.858,A -85,B 0,C 180,E1 22230.37,E2 22230.37} C_VEL
LIN {X 0,Y 464.139,Z 840.252,A -85,B 0,C 180,E1 22228.148,E2 22228.148} C_VEL
LIN {X 0,Y 464.123,Z 837.922,A -85,B 0,C 180,E1 22225.899,E2 22225.899} C_VEL
LIN {X 0,Y 464.127,Z 833.911,A -85,B 0,C 180,E1 22223.692,E2 22223.692} C_VEL
LIN {X 0,Y 464.181,Z 828.005,A -85,B 0,C 180,E1 22221.453,E2 22221.453} C_VEL
LIN {X 0,Y 464.332,Z 820.521,A -85,B 0,C 180,E1 22219.328,E2 22219.328} C_VEL
LIN {X 0,Y 464.63,Z 811.608,A -85,B 0,C 180,E1 22217.32,E2 22217.32} C_VEL
LIN {X 0,Y 465.096,Z 800.607,A -85,B 0,C 180,E1 22215.305,E2 22215.305} C_VEL
LIN {X 0,Y 465.843,Z 786.546,A -85,B 0,C 180,E1 22213.19,E2 22213.19} C_VEL
LIN {X 0,Y 466.676,Z 772.502,A -85,B 0,C 180,E1 22211.448,E2 22211.448} C_VEL
LIN {X 0,Y 467.597,Z 757.879,A -85,B 0,C 180,E1 22209.941,E2 22209.941} C_VEL
LIN {X 0,Y 468.592,Z 742.147,A -85,B 0,C 180,E1 22208.6,E2 22208.6} C_VEL
LIN {X 0,Y 469.577,Z 725.833,A -85,B 0,C 180,E1 22207.464,E2 22207.464} C_VEL
LIN {X 0,Y 470.541,Z 708.215,A -85,B 0,C 180,E1 22206.487,E2 22206.487} C_VEL
LIN {X 0,Y 471.405,Z 689.486,A -85,B 0,C 180,E1 22205.702,E2 22205.702} C_VEL
LIN {X 0,Y 472.117,Z 670.164,A -85,B 0,C 180,E1 22205.141,E2 22205.141} C_VEL
LIN {X 0,Y 472.586,Z 639.995,A -85,B 0,C 180,E1 22204.621,E2 22204.621} C_VEL
LIN {X 0,Y 473.296,Z 595.817,A -85,B 0,C 180,E1 22203.863,E2 22203.863} C_VEL
LIN {X 0,Y 476.198,Z 490.902,A -85,B 0,C 180,E1 22201.812,E2 22201.812} C_VEL
LIN {X 0,Y 476.322,Z 480.122,A -85,B 0,C 180,E1 22201.572,E2 22201.572} C_VEL
LIN {X 0,Y 473.179,Z 452.25,A -85,B 0,C 180,E1 22200.644,E2 22200.644} C_VEL
LIN {X 0,Y 476.1,Z 408.606,A -85,B 0,C 180,E1 22196.833,E2 22196.833} C_VEL
LIN {X 0,Y 476.492,Z 401.563,A -85,B 0,C 180,E1 22196.197,E2 22196.197} C_VEL
LIN {X 0,Y 468.138,Z 377.81,A -85,B 0,C 180,E1 22193.271,E2 22193.271} C_VEL
LIN {X 0,Y 464.96,Z 368.883,A -85,B 0,C 180,E1 22192.111,E2 22192.111} C_VEL
LIN {X 0,Y 464.942,Z 368.883,A -85,B 0,C 180,E1 22188.52,E2 22188.52} C_VEL
LIN {X 0,Y 464.947,Z 368.882,A -85,B 0,C 180,E1 22184.858,E2 22184.858} C_VEL
LIN {X 0,Y 464.987,Z 368.88,A -85,B 0,C 180,E1 22181.31,E2 22181.31} C_VEL
LIN {X 0,Y 464.968,Z 368.882,A -85,B 0,C 180,E1 22177.796,E2 22177.796} C_VEL
LIN {X 0,Y 464.968,Z 368.959,A -85,B 0,C 180,E1 22174.939,E2 22174.939} C_VEL
LIN {X 0,Y 465.923,Z 371.851,A -85,B 0,C 180,E1 22174.507,E2 22174.507} C_VEL
LIN {X 0,Y 467.23,Z 374.275,A -85,B 0,C 180,E1 22174.088,E2 22174.088} C_VEL
LIN {X 0,Y 471.348,Z 383.976,A -85,B 0,C 180,E1 22172.602,E2 22172.602} C_VEL
LIN {X 0,Y 475.554,Z 396.902,A -85,B 0,C 180,E1 22170.865,E2 22170.865} C_VEL
LIN {X 0,Y 476.489,Z 400.918,A -85,B 0,C 180,E1 22170.379,E2 22170.379} C_VEL
LIN {X 0,Y 476.126,Z 413.241,A -85,B 0,C 180,E1 22169.244,E2 22169.244} C_VEL
LIN {X 0,Y 478.385,Z 427.018,A -85,B 0,C 180,E1 22168.707,E2 22168.707} C_VEL
LIN {X 0,Y 474.881,Z 531.754,A -85,B 0,C 180,E1 22166.598,E2 22166.598} C_VEL
LIN {X 0,Y 472.941,Z 621.421,A -85,B 0,C 180,E1 22164.921,E2 22164.921} C_VEL
LIN {X 0,Y 472.322,Z 640.695,A -85,B 0,C 180,E1 22164.322,E2 22164.322} C_VEL
LIN {X 0,Y 471.575,Z 658.37,A -85,B 0,C 180,E1 22163.557,E2 22163.557} C_VEL
LIN {X 0,Y 470.633,Z 676.255,A -85,B 0,C 180,E1 22162.549,E2 22162.549} C_VEL
LIN {X 0,Y 469.563,Z 693.909,A -85,B 0,C 180,E1 22161.288,E2 22161.288} C_VEL
LIN {X 0,Y 468.52,Z 709.621,A -85,B 0,C 180,E1 22159.9,E2 22159.9} C_VEL
LIN {X 0,Y 467.489,Z 724.308,A -85,B 0,C 180,E1 22158.325,E2 22158.325} C_VEL
LIN {X 0,Y 466.53,Z 737.86,A -85,B 0,C 180,E1 22156.561,E2 22156.561} C_VEL
LIN {X 0,Y 465.714,Z 749.763,A -85,B 0,C 180,E1 22154.675,E2 22154.675} C_VEL
LIN {X 0,Y 465.066,Z 760.12,A -85,B 0,C 180,E1 22152.667,E2 22152.667} C_VEL
LIN {X 0,Y 464.609,Z 768.494,A -85,B 0,C 180,E1 22150.665,E2 22150.665} C_VEL
LIN {X 0,Y 464.296,Z 775.494,A -85,B 0,C 180,E1 22148.545,E2 22148.545} C_VEL
LIN {X 0,Y 464.108,Z 781.018,A -85,B 0,C 180,E1 22146.308,E2 22146.308} C_VEL
LIN {X 0,Y 464.017,Z 784.78,A -85,B 0,C 180,E1 22144.077,E2 22144.077} C_VEL
LIN {X 0,Y 463.986,Z 786.889,A -85,B 0,C 180,E1 22141.852,E2 22141.852} C_VEL
LIN {X 0,Y 463.987,Z 787.399,A -85,B 0,C 180,E1 22139.629,E2 22139.629} C_VEL
LIN {X 0,Y 463.989,Z 786.324,A -85,B 0,C 180,E1 22137.406,E2 22137.406} C_VEL
LIN {X 0,Y 464.027,Z 783.642,A -85,B 0,C 180,E1 22135.179,E2 22135.179} C_VEL
LIN {X 0,Y 464.133,Z 779.28,A -85,B 0,C 180,E1 22132.947,E2 22132.947} C_VEL
LIN {X 0,Y 464.348,Z 773.121,A -85,B 0,C 180,E1 22130.706,E2 22130.706} C_VEL
LIN {X 0,Y 464.726,Z 764.977,A -85,B 0,C 180,E1 22128.458,E2 22128.458} C_VEL
LIN {X 0,Y 465.283,Z 755.206,A -85,B 0,C 180,E1 22126.327,E2 22126.327} C_VEL
LIN {X 0,Y 465.981,Z 744.599,A -85,B 0,C 180,E1 22124.442,E2 22124.442} C_VEL
LIN {X 0,Y 466.831,Z 732.66,A -85,B 0,C 180,E1 22122.68,E2 22122.68} C_VEL
LIN {X 0,Y 467.832,Z 718.959,A -85,B 0,C 180,E1 22120.996,E2 22120.996} C_VEL
LIN {X 0,Y 468.929,Z 703.936,A -85,B 0,C 180,E1 22119.467,E2 22119.467} C_VEL
LIN {X 0,Y 470.075,Z 687.345,A -85,B 0,C 180,E1 22118.081,E2 22118.081} C_VEL
LIN {X 0,Y 471.126,Z 670.517,A -85,B 0,C 180,E1 22116.948,E2 22116.948} C_VEL
LIN {X 0,Y 472.075,Z 652.78,A -85,B 0,C 180,E1 22116.005,E2 22116.005} C_VEL
LIN {X 0,Y 472.882,Z 634.178,A -85,B 0,C 180,E1 22115.259,E2 22115.259} C_VEL
LIN {X 0,Y 473.483,Z 615.145,A -85,B 0,C 180,E1 22114.729,E2 22114.729} C_VEL
LIN {X 0,Y 477.018,Z 425.119,A -85,B 0,C 180,E1 22111.425,E2 22111.425} C_VEL
LIN {X 0,Y 473.745,Z 407.211,A -85,B 0,C 180,E1 22110.859,E2 22110.859} C_VEL
LIN {X 0,Y 473.963,Z 397.133,A -85,B 0,C 180,E1 22109.862,E2 22109.862} C_VEL
LIN {X 0,Y 467.651,Z 377.14,A -85,B 0,C 180,E1 22107.394,E2 22107.394} C_VEL
LIN {X 0,Y 464.984,Z 368.876,A -85,B 0,C 180,E1 22106.323,E2 22106.323} C_VEL
LIN {X 0,Y 464.993,Z 368.876,A -85,B 0,C 180,E1 22102.672,E2 22102.672} C_VEL
LIN {X 0,Y 464.945,Z 368.881,A -85,B 0,C 180,E1 22101.484,E2 22101.484} C_VEL
LIN {X 0,Y 463.952,Z 369.005,A -85,B 0,C 180,E1 22100.534,E2 22100.534} C_VEL
LIN {X 0,Y 457.519,Z 369.808,A -85,B 0,C 180,E1 22097.862,E2 22097.862} C_VEL
LIN {X 0,Y 457.012,Z 369.869,A -85,B 0,C 180,E1 22097.165,E2 22097.165} C_VEL
LIN {X 0,Y 457.006,Z 369.868,A -85,B 0,C 180,E1 22093.565,E2 22093.565} C_VEL
LIN {X 0,Y 457.032,Z 369.868,A -85,B 0,C 180,E1 22090.03,E2 22090.03} C_VEL
LIN {X 0,Y 457.051,Z 369.868,A -85,B 0,C 180,E1 22086.515,E2 22086.515} C_VEL
LIN {X 0,Y 457.01,Z 369.869,A -85,B 0,C 180,E1 22083.009,E2 22083.009} C_VEL
LIN {X 0,Y 457.004,Z 369.867,A -85,B 0,C 180,E1 22079.346,E2 22079.346} C_VEL
LIN {X 0,Y 457.027,Z 369.868,A -85,B 0,C 180,E1 22075.808,E2 22075.808} C_VEL
LIN {X 0,Y 457.067,Z 369.866,A -85,B 0,C 180,E1 22072.238,E2 22072.238} C_VEL
LIN {X 0,Y 457.023,Z 369.868,A -85,B 0,C 180,E1 22068.628,E2 22068.628} C_VEL
LIN {X 0,Y 457.001,Z 369.869,A -85,B 0,C 180,E1 22065.091,E2 22065.091} C_VEL
LIN {X 0,Y 457.012,Z 369.868,A -85,B 0,C 180,E1 22061.436,E2 22061.436} C_VEL
LIN {X 0,Y 457.056,Z 369.866,A -85,B 0,C 180,E1 22057.922,E2 22057.922} C_VEL
LIN {X 0,Y 457.039,Z 369.866,A -85,B 0,C 180,E1 22054.266,E2 22054.266} C_VEL
LIN {X 0,Y 457.003,Z 369.867,A -85,B 0,C 180,E1 22050.752,E2 22050.752} C_VEL
LIN {X 0,Y 457.005,Z 369.865,A -85,B 0,C 180,E1 22047.116,E2 22047.116} C_VEL
LIN {X 0,Y 457.036,Z 369.865,A -85,B 0,C 180,E1 22043.594,E2 22043.594} C_VEL
LIN {X 0,Y 457.045,Z 369.866,A -85,B 0,C 180,E1 22040.048,E2 22040.048} C_VEL
LIN {X 0,Y 457.009,Z 369.866,A -85,B 0,C 180,E1 22036.461,E2 22036.461} C_VEL
LIN {X 0,Y 457.002,Z 369.867,A -85,B 0,C 180,E1 22032.821,E2 22032.821} C_VEL
LIN {X 0,Y 457.019,Z 369.867,A -85,B 0,C 180,E1 22029.242,E2 22029.242} C_VEL
LIN {X 0,Y 457.055,Z 369.866,A -85,B 0,C 180,E1 22025.715,E2 22025.715} C_VEL
LIN {X 0,Y 457.024,Z 369.867,A -85,B 0,C 180,E1 22022.083,E2 22022.083} C_VEL
LIN {X 0,Y 457.001,Z 369.869,A -85,B 0,C 180,E1 22018.57,E2 22018.57} C_VEL
LIN {X 0,Y 457.005,Z 369.871,A -85,B 0,C 180,E1 22014.872,E2 22014.872} C_VEL
LIN {X 0,Y 457.037,Z 369.871,A -85,B 0,C 180,E1 22011.267,E2 22011.267} C_VEL
LIN {X 0,Y 457.049,Z 369.868,A -85,B 0,C 180,E1 22007.639,E2 22007.639} C_VEL
LIN {X 0,Y 457.011,Z 369.869,A -85,B 0,C 180,E1 22004.086,E2 22004.086} C_VEL
LIN {X 0,Y 457,Z 369.871,A -85,B 0,C 180,E1 22000.527,E2 22000.527} C_VEL
LIN {X 0,Y 457.025,Z 369.872,A -85,B 0,C 180,E1 21996.987,E2 21996.987} C_VEL
LIN {X 0,Y 457.053,Z 369.868,A -85,B 0,C 180,E1 21993.455,E2 21993.455} C_VEL
LIN {X 0,Y 457.058,Z 370.026,A -85,B 0,C 180,E1 21993.086,E2 21993.086} C_VEL
LIN {X 0,Y 462.535,Z 390.24,A -85,B 0,C 180,E1 21989.814,E2 21989.814} C_VEL
LIN {X 0,Y 463.834,Z 396.346,A -85,B 0,C 180,E1 21988.873,E2 21988.873} C_VEL
LIN {X 0,Y 462.164,Z 424.116,A -85,B 0,C 180,E1 21985.158,E2 21985.158} C_VEL
LIN {X 0,Y 460.625,Z 452.711,A -85,B 0,C 180,E1 21981.387,E2 21981.387} C_VEL
LIN {X 0,Y 459.449,Z 479.672,A -85,B 0,C 180,E1 21977.915,E2 21977.915} C_VEL
LIN {X 0,Y 462.034,Z 498.087,A -85,B 0,C 180,E1 21977.439,E2 21977.439} C_VEL
LIN {X 0,Y 460.294,Z 599.375,A -85,B 0,C 180,E1 21975.533,E2 21975.533} C_VEL
LIN {X 0,Y 459.996,Z 614.624,A -85,B 0,C 180,E1 21975.023,E2 21975.023} C_VEL
LIN {X 0,Y 459.571,Z 629.809,A -85,B 0,C 180,E1 21974.272,E2 21974.272} C_VEL
LIN {X 0,Y 459.006,Z 644.357,A -85,B 0,C 180,E1 21973.286,E2 21973.286} C_VEL
LIN {X 0,Y 458.504,Z 656.607,A -85,B 0,C 180,E1 21972.212,E2 21972.212} C_VEL
LIN {X 0,Y 458.012,Z 668.58,A -85,B 0,C 180,E1 21970.885,E2 21970.885} C_VEL
LIN {X 0,Y 457.535,Z 679.676,A -85,B 0,C 180,E1 21969.307,E2 21969.307} C_VEL
LIN {X 0,Y 457.18,Z 688.556,A -85,B 0,C 180,E1 21967.667,E2 21967.667} C_VEL
LIN {X 0,Y 456.947,Z 695.368,A -85,B 0,C 180,E1 21966.029,E2 21966.029} C_VEL
LIN {X 0,Y 456.805,Z 700.738,A -85,B 0,C 180,E1 21964.268,E2 21964.268} C_VEL
LIN {X 0,Y 456.734,Z 704.263,A -85,B 0,C 180,E1 21962.51,E2 21962.51} C_VEL
LIN {X 0,Y 456.754,Z 706.237,A -85,B 0,C 180,E1 21960.627,E2 21960.627} C_VEL
LIN {X 0,Y 456.797,Z 706.317,A -85,B 0,C 180,E1 21958.746,E2 21958.746} C_VEL
LIN {X 0,Y 456.915,Z 704.711,A -85,B 0,C 180,E1 21956.99,E2 21956.99} C_VEL
LIN {X 0,Y 457.109,Z 701.117,A -85,B 0,C 180,E1 21955.106,E2 21955.106} C_VEL
LIN {X 0,Y 457.389,Z 695.802,A -85,B 0,C 180,E1 21953.347,E2 21953.347} C_VEL
LIN {X 0,Y 457.76,Z 688.876,A -85,B 0,C 180,E1 21951.677,E2 21951.677} C_VEL
LIN {X 0,Y 458.237,Z 680.107,A -85,B 0,C 180,E1 21950.074,E2 21950.074} C_VEL
LIN {X 0,Y 458.796,Z 669.871,A -85,B 0,C 180,E1 21948.625,E2 21948.625} C_VEL
LIN {X 0,Y 459.374,Z 658.642,A -85,B 0,C 180,E1 21947.365,E2 21947.365} C_VEL
LIN {X 0,Y 460.011,Z 644.983,A -85,B 0,C 180,E1 21946.167,E2 21946.167} C_VEL
LIN {X 0,Y 460.659,Z 629.816,A -85,B 0,C 180,E1 21945.16,E2 21945.16} C_VEL
LIN {X 0,Y 461.168,Z 614.156,A -85,B 0,C 180,E1 21944.405,E2 21944.405} C_VEL
LIN {X 0,Y 461.542,Z 598.205,A -85,B 0,C 180,E1 21943.889,E2 21943.889} C_VEL
LIN {X 0,Y 465.067,Z 501.594,A -85,B 0,C 180,E1 21941.609,E2 21941.609} C_VEL
LIN {X 0,Y 464.947,Z 497.061,A -85,B 0,C 180,E1 21941.473,E2 21941.473} C_VEL
LIN {X 0,Y 461.742,Z 479.332,A -85,B 0,C 180,E1 21940.716,E2 21940.716} C_VEL
LIN {X 0,Y 463.936,Z 450.799,A -85,B 0,C 180,E1 21936.772,E2 21936.772} C_VEL
LIN {X 0,Y 466.521,Z 424.388,A -85,B 0,C 180,E1 21932.976,E2 21932.976} C_VEL
LIN {X 0,Y 468.85,Z 404.949,A -85,B 0,C 180,E1 21930.065,E2 21930.065} C_VEL
LIN {X 0,Y 466.35,Z 394.644,A -85,B 0,C 180,E1 21927.875,E2 21927.875} C_VEL
LIN {X 0,Y 463.328,Z 385.141,A -85,B 0,C 180,E1 21925.42,E2 21925.42} C_VEL
LIN {X 0,Y 461.42,Z 380.518,A -85,B 0,C 180,E1 21923.927,E2 21923.927} C_VEL
LIN {X 0,Y 460.302,Z 377.622,A -85,B 0,C 180,E1 21922.853,E2 21922.853} C_VEL
LIN {X 0,Y 458.889,Z 374.113,A -85,B 0,C 180,E1 21921.264,E2 21921.264} C_VEL
LIN {X 0,Y 457.24,Z 370.935,A -85,B 0,C 180,E1 21918.837,E2 21918.837} C_VEL
LIN {X 0,Y 457.023,Z 369.871,A -85,B 0,C 180,E1 21916.947,E2 21916.947} C_VEL
LIN {X 0,Y 457.1,Z 370.463,A -85,B 0,C 180,E1 21915.309,E2 21915.309} C_VEL
LIN {X 0,Y 458.281,Z 373.297,A -85,B 0,C 180,E1 21913.039,E2 21913.039} C_VEL
LIN {X 0,Y 459.471,Z 375.135,A -85,B 0,C 180,E1 21912,E2 21912} C_VEL
LIN {X 0,Y 461.225,Z 378.743,A -85,B 0,C 180,E1 21910.568,E2 21910.568} C_VEL
LIN {X 0,Y 463.743,Z 384.882,A -85,B 0,C 180,E1 21908.793,E2 21908.793} C_VEL
LIN {X 0,Y 466.924,Z 392.683,A -85,B 0,C 180,E1 21906.991,E2 21906.991} C_VEL
LIN {X 0,Y 470.17,Z 402.531,A -85,B 0,C 180,E1 21905.191,E2 21905.191} C_VEL
LIN {X 0,Y 471.559,Z 407.295,A -85,B 0,C 180,E1 21904.431,E2 21904.431} C_VEL
LIN {X 0,Y 467.696,Z 438.274,A -85,B 0,C 180,E1 21901.299,E2 21901.299} C_VEL
LIN {X 0,Y 465.88,Z 459.236,A -85,B 0,C 180,E1 21899.342,E2 21899.342} C_VEL
LIN {X 0,Y 468.835,Z 484.056,A -85,B 0,C 180,E1 21898.662,E2 21898.662} C_VEL
LIN {X 0,Y 465.079,Z 670.079,A -85,B 0,C 180,E1 21895.343,E2 21895.343} C_VEL
LIN {X 0,Y 464.312,Z 689.068,A -85,B 0,C 180,E1 21894.783,E2 21894.783} C_VEL
LIN {X 0,Y 463.401,Z 707.205,A -85,B 0,C 180,E1 21894.022,E2 21894.022} C_VEL
LIN {X 0,Y 462.337,Z 724.927,A -85,B 0,C 180,E1 21893.044,E2 21893.044} C_VEL
LIN {X 0,Y 461.189,Z 742.314,A -85,B 0,C 180,E1 21891.828,E2 21891.828} C_VEL
LIN {X 0,Y 460.052,Z 758.64,A -85,B 0,C 180,E1 21890.416,E2 21890.416} C_VEL
LIN {X 0,Y 459.027,Z 773.333,A -85,B 0,C 180,E1 21888.873,E2 21888.873} C_VEL
LIN {X 0,Y 458.104,Z 787.078,A -85,B 0,C 180,E1 21887.137,E2 21887.137} C_VEL
LIN {X 0,Y 457.322,Z 799.721,A -85,B 0,C 180,E1 21885.21,E2 21885.21} C_VEL
LIN {X 0,Y 456.767,Z 810.751,A -85,B 0,C 180,E1 21883.159,E2 21883.159} C_VEL
LIN {X 0,Y 456.369,Z 820.159,A -85,B 0,C 180,E1 21880.988,E2 21880.988} C_VEL
LIN {X 0,Y 456.182,Z 827.569,A -85,B 0,C 180,E1 21878.826,E2 21878.826} C_VEL
LIN {X 0,Y 456.121,Z 833.196,A -85,B 0,C 180,E1 21876.672,E2 21876.672} C_VEL
LIN {X 0,Y 456.114,Z 837.341,A -85,B 0,C 180,E1 21874.4,E2 21874.4} C_VEL
LIN {X 0,Y 456.142,Z 839.737,A -85,B 0,C 180,E1 21872.136,E2 21872.136} C_VEL
LIN {X 0,Y 456.162,Z 840.438,A -85,B 0,C 180,E1 21869.874,E2 21869.874} C_VEL
LIN {X 0,Y 456.145,Z 839.446,A -85,B 0,C 180,E1 21867.613,E2 21867.613} C_VEL
LIN {X 0,Y 456.126,Z 836.738,A -85,B 0,C 180,E1 21865.348,E2 21865.348} C_VEL
LIN {X 0,Y 456.14,Z 832.236,A -85,B 0,C 180,E1 21863.076,E2 21863.076} C_VEL
LIN {X 0,Y 456.207,Z 826.236,A -85,B 0,C 180,E1 21860.921,E2 21860.921} C_VEL
LIN {X 0,Y 456.402,Z 818.346,A -85,B 0,C 180,E1 21858.757,E2 21858.757} C_VEL
LIN {X 0,Y 456.756,Z 808.991,A -85,B 0,C 180,E1 21856.712,E2 21856.712} C_VEL
LIN {X 0,Y 457.254,Z 798.234,A -85,B 0,C 180,E1 21854.787,E2 21854.787} C_VEL
LIN {X 0,Y 457.991,Z 785.151,A -85,B 0,C 180,E1 21852.859,E2 21852.859} C_VEL
LIN {X 0,Y 458.979,Z 769.27,A -85,B 0,C 180,E1 21850.927,E2 21850.927} C_VEL
LIN {X 0,Y 460.05,Z 753.27,A -85,B 0,C 180,E1 21849.318,E2 21849.318} C_VEL
LIN {X 0,Y 461.136,Z 736.902,A -85,B 0,C 180,E1 21847.969,E2 21847.969} C_VEL
LIN {X 0,Y 462.219,Z 719.479,A -85,B 0,C 180,E1 21846.815,E2 21846.815} C_VEL
LIN {X 0,Y 463.213,Z 701.524,A -85,B 0,C 180,E1 21845.889,E2 21845.889} C_VEL
LIN {X 0,Y 464.091,Z 682.554,A -85,B 0,C 180,E1 21845.167,E2 21845.167} C_VEL
LIN {X 0,Y 464.721,Z 663.3,A -85,B 0,C 180,E1 21844.679,E2 21844.679} C_VEL
LIN {X 0,Y 466.894,Z 566.61,A -85,B 0,C 180,E1 21842.857,E2 21842.857} C_VEL
LIN {X 0,Y 469.595,Z 481.636,A -85,B 0,C 180,E1 21841.079,E2 21841.079} C_VEL
LIN {X 0,Y 466.565,Z 453.431,A -85,B 0,C 180,E1 21840.091,E2 21840.091} C_VEL
LIN {X 0,Y 466.056,Z 448.197,A -85,B 0,C 180,E1 21839.866,E2 21839.866} C_VEL
LIN {X 0,Y 469.257,Z 404.648,A -85,B 0,C 180,E1 21835.981,E2 21835.981} C_VEL
LIN {X 0,Y 461.254,Z 381.715,A -85,B 0,C 180,E1 21833.119,E2 21833.119} C_VEL
LIN {X 0,Y 457.062,Z 369.862,A -85,B 0,C 180,E1 21831.55,E2 21831.55} C_VEL
LIN {X 0,Y 457.028,Z 369.87,A -85,B 0,C 180,E1 21827.975,E2 21827.975} C_VEL
LIN {X 0,Y 457.003,Z 369.872,A -85,B 0,C 180,E1 21824.436,E2 21824.436} C_VEL
LIN {X 0,Y 457.004,Z 369.872,A -85,B 0,C 180,E1 21820.691,E2 21820.691} C_VEL
LIN {X 0,Y 457.034,Z 369.87,A -85,B 0,C 180,E1 21817.143,E2 21817.143} C_VEL
LIN {X 0,Y 457.027,Z 369.982,A -85,B 0,C 180,E1 21815.993,E2 21815.993} C_VEL
LIN {X 0,Y 458.127,Z 372.991,A -85,B 0,C 180,E1 21815.489,E2 21815.489} C_VEL
LIN {X 0,Y 459.377,Z 375.086,A -85,B 0,C 180,E1 21815.072,E2 21815.072} C_VEL
LIN {X 0,Y 464.088,Z 385.827,A -85,B 0,C 180,E1 21813.287,E2 21813.287} C_VEL
LIN {X 0,Y 468.04,Z 397.242,A -85,B 0,C 180,E1 21811.646,E2 21811.646} C_VEL
LIN {X 0,Y 469.831,Z 404.699,A -85,B 0,C 180,E1 21810.709,E2 21810.709} C_VEL
LIN {X 0,Y 469.472,Z 414.065,A -85,B 0,C 180,E1 21809.833,E2 21809.833} C_VEL
LIN {X 0,Y 471.796,Z 428.182,A -85,B 0,C 180,E1 21809.241,E2 21809.241} C_VEL
LIN {X 0,Y 467.888,Z 531.524,A -85,B 0,C 180,E1 21807.076,E2 21807.076} C_VEL
LIN {X 0,Y 465.638,Z 622.203,A -85,B 0,C 180,E1 21805.309,E2 21805.309} C_VEL
LIN {X 0,Y 464.966,Z 641.487,A -85,B 0,C 180,E1 21804.694,E2 21804.694} C_VEL
LIN {X 0,Y 464.136,Z 659.56,A -85,B 0,C 180,E1 21803.891,E2 21803.891} C_VEL
LIN {X 0,Y 463.134,Z 677.268,A -85,B 0,C 180,E1 21802.867,E2 21802.867} C_VEL
LIN {X 0,Y 461.993,Z 694.802,A -85,B 0,C 180,E1 21801.587,E2 21801.587} C_VEL
LIN {X 0,Y 460.881,Z 710.443,A -85,B 0,C 180,E1 21800.178,E2 21800.178} C_VEL
LIN {X 0,Y 459.776,Z 725.13,A -85,B 0,C 180,E1 21798.571,E2 21798.571} C_VEL
LIN {X 0,Y 458.787,Z 738.14,A -85,B 0,C 180,E1 21796.849,E2 21796.849} C_VEL
LIN {X 0,Y 457.903,Z 750.1,A -85,B 0,C 180,E1 21794.931,E2 21794.931} C_VEL
LIN {X 0,Y 457.196,Z 760.492,A -85,B 0,C 180,E1 21792.889,E2 21792.889} C_VEL
LIN {X 0,Y 456.695,Z 768.9,A -85,B 0,C 180,E1 21790.852,E2 21790.852} C_VEL
LIN {X 0,Y 456.349,Z 775.924,A -85,B 0,C 180,E1 21788.695,E2 21788.695} C_VEL
LIN {X 0,Y 456.139,Z 781.471,A -85,B 0,C 180,E1 21786.418,E2 21786.418} C_VEL
LIN {X 0,Y 456.037,Z 785.246,A -85,B 0,C 180,E1 21784.149,E2 21784.149} C_VEL
LIN {X 0,Y 456.001,Z 787.357,A -85,B 0,C 180,E1 21781.885,E2 21781.885} C_VEL
LIN {X 0,Y 456.001,Z 787.858,A -85,B 0,C 180,E1 21779.623,E2 21779.623} C_VEL
LIN {X 0,Y 456.004,Z 786.763,A -85,B 0,C 180,E1 21777.361,E2 21777.361} C_VEL
LIN {X 0,Y 456.048,Z 784.052,A -85,B 0,C 180,E1 21775.095,E2 21775.095} C_VEL
LIN {X 0,Y 456.165,Z 779.65,A -85,B 0,C 180,E1 21772.823,E2 21772.823} C_VEL
LIN {X 0,Y 456.401,Z 773.44,A -85,B 0,C 180,E1 21770.543,E2 21770.543} C_VEL
LIN {X 0,Y 456.817,Z 765.239,A -85,B 0,C 180,E1 21768.255,E2 21768.255} C_VEL
LIN {X 0,Y 457.419,Z 755.398,A -85,B 0,C 180,E1 21766.087,E2 21766.087} C_VEL
LIN {X 0,Y 458.17,Z 744.711,A -85,B 0,C 180,E1 21764.17,E2 21764.17} C_VEL
LIN {X 0,Y 459.08,Z 732.685,A -85,B 0,C 180,E1 21762.378,E2 21762.378} C_VEL
LIN {X 0,Y 460.17,Z 718.731,A -85,B 0,C 180,E1 21760.649,E2 21760.649} C_VEL
LIN {X 0,Y 461.353,Z 703.393,A -85,B 0,C 180,E1 21759.08,E2 21759.08} C_VEL
LIN {X 0,Y 462.545,Z 686.804,A -85,B 0,C 180,E1 21757.697,E2 21757.697} C_VEL
LIN {X 0,Y 463.678,Z 669.436,A -85,B 0,C 180,E1 21756.531,E2 21756.531} C_VEL
LIN {X 0,Y 464.662,Z 651.786,A -85,B 0,C 180,E1 21755.597,E2 21755.597} C_VEL
LIN {X 0,Y 465.495,Z 632.992,A -85,B 0,C 180,E1 21754.85,E2 21754.85} C_VEL
LIN {X 0,Y 466.133,Z 613.349,A -85,B 0,C 180,E1 21754.315,E2 21754.315} C_VEL
LIN {X 0,Y 469.906,Z 426.406,A -85,B 0,C 180,E1 21750.997,E2 21750.997} C_VEL
LIN {X 0,Y 466.497,Z 407.589,A -85,B 0,C 180,E1 21750.392,E2 21750.392} C_VEL
LIN {X 0,Y 466.66,Z 399.891,A -85,B 0,C 180,E1 21749.625,E2 21749.625} C_VEL
LIN {X 0,Y 460.455,Z 380.289,A -85,B 0,C 180,E1 21747.178,E2 21747.178} C_VEL
LIN {X 0,Y 457.01,Z 369.869,A -85,B 0,C 180,E1 21745.827,E2 21745.827} C_VEL
LIN {X 0,Y 457.039,Z 369.866,A -85,B 0,C 180,E1 21742.225,E2 21742.225} C_VEL
LIN {X 0,Y 457.058,Z 369.867,A -85,B 0,C 180,E1 21738.621,E2 21738.621} C_VEL
LIN {X 0,Y 457.012,Z 369.869,A -85,B 0,C 180,E1 21737.165,E2 21737.165} C_VEL
LIN {X 0,Y 456.039,Z 369.993,A -85,B 0,C 180,E1 21736.198,E2 21736.198} C_VEL
LIN {X 0,Y 449.583,Z 370.795,A -85,B 0,C 180,E1 21733.48,E2 21733.48} C_VEL
LIN {X 0,Y 449.096,Z 370.856,A -85,B 0,C 180,E1 21732.77,E2 21732.77} C_VEL
LIN {X 0,Y 449.067,Z 370.857,A -85,B 0,C 180,E1 21729.21,E2 21729.21} C_VEL
LIN {X 0,Y 449.065,Z 370.858,A -85,B 0,C 180,E1 21725.421,E2 21725.421} C_VEL
LIN {X 0,Y 449.079,Z 370.858,A -85,B 0,C 180,E1 21721.732,E2 21721.732} C_VEL
LIN {X 0,Y 449.121,Z 370.857,A -85,B 0,C 180,E1 21718.162,E2 21718.162} C_VEL
LIN {X 0,Y 449.11,Z 370.856,A -85,B 0,C 180,E1 21714.416,E2 21714.416} C_VEL
LIN {X 0,Y 449.072,Z 370.855,A -85,B 0,C 180,E1 21710.87,E2 21710.87} C_VEL
LIN {X 0,Y 449.066,Z 370.853,A -85,B 0,C 180,E1 21707.218,E2 21707.218} C_VEL
LIN {X 0,Y 449.086,Z 370.854,A -85,B 0,C 180,E1 21703.651,E2 21703.651} C_VEL
LIN {X 0,Y 449.115,Z 370.855,A -85,B 0,C 180,E1 21700,E2 21700} C_VEL
LIN {X 0,Y 449.09,Z 370.856,A -85,B 0,C 180,E1 21696.391,E2 21696.391} C_VEL
LIN {X 0,Y 449.064,Z 370.853,A -85,B 0,C 180,E1 21692.808,E2 21692.808} C_VEL
LIN {X 0,Y 449.064,Z 370.853,A -85,B 0,C 180,E1 21689.107,E2 21689.107} C_VEL
LIN {X 0,Y 449.088,Z 370.857,A -85,B 0,C 180,E1 21685.531,E2 21685.531} C_VEL
LIN {X 0,Y 449.121,Z 370.851,A -85,B 0,C 180,E1 21681.937,E2 21681.937} C_VEL
LIN {X 0,Y 449.091,Z 370.856,A -85,B 0,C 180,E1 21678.18,E2 21678.18} C_VEL
LIN {X 0,Y 449.063,Z 370.858,A -85,B 0,C 180,E1 21674.635,E2 21674.635} C_VEL
LIN {X 0,Y 449.066,Z 370.858,A -85,B 0,C 180,E1 21670.895,E2 21670.895} C_VEL
LIN {X 0,Y 449.091,Z 370.857,A -85,B 0,C 180,E1 21667.346,E2 21667.346} C_VEL
LIN {X 0,Y 449.116,Z 370.856,A -85,B 0,C 180,E1 21663.702,E2 21663.702} C_VEL
LIN {X 0,Y 449.082,Z 370.856,A -85,B 0,C 180,E1 21660.084,E2 21660.084} C_VEL
LIN {X 0,Y 449.062,Z 370.86,A -85,B 0,C 180,E1 21656.483,E2 21656.483} C_VEL
LIN {X 0,Y 449.064,Z 370.86,A -85,B 0,C 180,E1 21652.726,E2 21652.726} C_VEL
LIN {X 0,Y 449.093,Z 370.857,A -85,B 0,C 180,E1 21649.199,E2 21649.199} C_VEL
LIN {X 0,Y 449.114,Z 370.856,A -85,B 0,C 180,E1 21645.47,E2 21645.47} C_VEL
LIN {X 0,Y 449.095,Z 370.859,A -85,B 0,C 180,E1 21641.736,E2 21641.736} C_VEL
LIN {X 0,Y 449.063,Z 370.86,A -85,B 0,C 180,E1 21638.189,E2 21638.189} C_VEL
LIN {X 0,Y 449.061,Z 370.862,A -85,B 0,C 180,E1 21634.44,E2 21634.44} C_VEL
LIN {X 0,Y 449.135,Z 371.067,A -85,B 0,C 180,E1 21633.538,E2 21633.538} C_VEL
LIN {X 0,Y 454.656,Z 391.263,A -85,B 0,C 180,E1 21630.2,E2 21630.2} C_VEL
LIN {X 0,Y 456.282,Z 398.189,A -85,B 0,C 180,E1 21629.109,E2 21629.109} C_VEL
LIN {X 0,Y 454.534,Z 425.55,A -85,B 0,C 180,E1 21625.401,E2 21625.401} C_VEL
LIN {X 0,Y 452.927,Z 453.75,A -85,B 0,C 180,E1 21621.633,E2 21621.633} C_VEL
LIN {X 0,Y 451.724,Z 479.626,A -85,B 0,C 180,E1 21618.261,E2 21618.261} C_VEL
LIN {X 0,Y 454.435,Z 498.971,A -85,B 0,C 180,E1 21617.742,E2 21617.742} C_VEL
LIN {X 0,Y 452.57,Z 600.067,A -85,B 0,C 180,E1 21615.785,E2 21615.785} C_VEL
LIN {X 0,Y 452.248,Z 615.504,A -85,B 0,C 180,E1 21615.254,E2 21615.254} C_VEL
LIN {X 0,Y 451.797,Z 630.768,A -85,B 0,C 180,E1 21614.482,E2 21614.482} C_VEL
LIN {X 0,Y 451.194,Z 645.611,A -85,B 0,C 180,E1 21613.455,E2 21613.455} C_VEL
LIN {X 0,Y 450.643,Z 658.408,A -85,B 0,C 180,E1 21612.298,E2 21612.298} C_VEL
LIN {X 0,Y 450.152,Z 669.727,A -85,B 0,C 180,E1 21611.012,E2 21611.012} C_VEL
LIN {X 0,Y 449.67,Z 680.441,A -85,B 0,C 180,E1 21609.471,E2 21609.471} C_VEL
LIN {X 0,Y 449.294,Z 689.427,A -85,B 0,C 180,E1 21607.802,E2 21607.802} C_VEL
LIN {X 0,Y 449.045,Z 696.327,A -85,B 0,C 180,E1 21606.136,E2 21606.136} C_VEL
LIN {X 0,Y 448.893,Z 701.78,A -85,B 0,C 180,E1 21604.343,E2 21604.343} C_VEL
LIN {X 0,Y 448.819,Z 705.378,A -85,B 0,C 180,E1 21602.554,E2 21602.554} C_VEL
LIN {X 0,Y 448.842,Z 707.422,A -85,B 0,C 180,E1 21600.638,E2 21600.638} C_VEL
LIN {X 0,Y 448.895,Z 707.553,A -85,B 0,C 180,E1 21598.724,E2 21598.724} C_VEL
LIN {X 0,Y 449.029,Z 705.992,A -85,B 0,C 180,E1 21596.937,E2 21596.937} C_VEL
LIN {X 0,Y 449.249,Z 702.448,A -85,B 0,C 180,E1 21595.021,E2 21595.021} C_VEL
LIN {X 0,Y 449.564,Z 697.192,A -85,B 0,C 180,E1 21593.231,E2 21593.231} C_VEL
LIN {X 0,Y 449.967,Z 690.478,A -85,B 0,C 180,E1 21591.567,E2 21591.567} C_VEL
LIN {X 0,Y 450.489,Z 681.559,A -85,B 0,C 180,E1 21589.902,E2 21589.902} C_VEL
LIN {X 0,Y 451.084,Z 671.497,A -85,B 0,C 180,E1 21588.445,E2 21588.445} C_VEL
LIN {X 0,Y 451.724,Z 660.295,A -85,B 0,C 180,E1 21587.147,E2 21587.147} C_VEL
LIN {X 0,Y 452.41,Z 646.846,A -85,B 0,C 180,E1 21585.93,E2 21585.93} C_VEL
LIN {X 0,Y 453.054,Z 633.025,A -85,B 0,C 180,E1 21584.971,E2 21584.971} C_VEL
LIN {X 0,Y 453.596,Z 618.364,A -85,B 0,C 180,E1 21584.203,E2 21584.203} C_VEL
LIN {X 0,Y 454.058,Z 601.99,A -85,B 0,C 180,E1 21583.608,E2 21583.608} C_VEL
LIN {X 0,Y 458.098,Z 501.481,A -85,B 0,C 180,E1 21581.117,E2 21581.117} C_VEL
LIN {X 0,Y 457.486,Z 495.626,A -85,B 0,C 180,E1 21580.899,E2 21580.899} C_VEL
LIN {X 0,Y 454.463,Z 479.336,A -85,B 0,C 180,E1 21580.162,E2 21580.162} C_VEL
LIN {X 0,Y 456.925,Z 450.742,A -85,B 0,C 180,E1 21576.12,E2 21576.12} C_VEL
LIN {X 0,Y 459.858,Z 424.466,A -85,B 0,C 180,E1 21572.244,E2 21572.244} C_VEL
LIN {X 0,Y 461.935,Z 408.144,A -85,B 0,C 180,E1 21569.713,E2 21569.713} C_VEL
LIN {X 0,Y 459.606,Z 398.215,A -85,B 0,C 180,E1 21567.497,E2 21567.497} C_VEL
LIN {X 0,Y 457.138,Z 390.171,A -85,B 0,C 180,E1 21565.326,E2 21565.326} C_VEL
LIN {X 0,Y 454.779,Z 383.577,A -85,B 0,C 180,E1 21563.052,E2 21563.052} C_VEL
LIN {X 0,Y 452.943,Z 379.393,A -85,B 0,C 180,E1 21560.99,E2 21560.99} C_VEL
LIN {X 0,Y 451.679,Z 376.326,A -85,B 0,C 180,E1 21558.387,E2 21558.387} C_VEL
LIN {X 0,Y 451.653,Z 375.781,A -85,B 0,C 180,E1 21556.315,E2 21556.315} C_VEL
LIN {X 0,Y 452.072,Z 377.572,A -85,B 0,C 180,E1 21554.226,E2 21554.226} C_VEL
LIN {X 0,Y 453.831,Z 380.536,A -85,B 0,C 180,E1 21552.219,E2 21552.219} C_VEL
LIN {X 0,Y 455.413,Z 384.166,A -85,B 0,C 180,E1 21550.76,E2 21550.76} C_VEL
LIN {X 0,Y 457.929,Z 390.357,A -85,B 0,C 180,E1 21548.886,E2 21548.886} C_VEL
LIN {X 0,Y 460.932,Z 398.263,A -85,B 0,C 180,E1 21547.035,E2 21547.035} C_VEL
LIN {X 0,Y 463.727,Z 406.926,A -85,B 0,C 180,E1 21545.411,E2 21545.411} C_VEL
LIN {X 0,Y 464.704,Z 411.298,A -85,B 0,C 180,E1 21544.723,E2 21544.723} C_VEL
LIN {X 0,Y 460.504,Z 441.821,A -85,B 0,C 180,E1 21541.552,E2 21541.552} C_VEL
LIN {X 0,Y 458.764,Z 460.159,A -85,B 0,C 180,E1 21539.797,E2 21539.797} C_VEL
LIN {X 0,Y 461.709,Z 484.999,A -85,B 0,C 180,E1 21539.1,E2 21539.1} C_VEL
LIN {X 0,Y 457.657,Z 669.886,A -85,B 0,C 180,E1 21535.718,E2 21535.718} C_VEL
LIN {X 0,Y 456.836,Z 688.963,A -85,B 0,C 180,E1 21535.143,E2 21535.143} C_VEL
LIN {X 0,Y 455.846,Z 707.346,A -85,B 0,C 180,E1 21534.353,E2 21534.353} C_VEL
LIN {X 0,Y 454.674,Z 725.606,A -85,B 0,C 180,E1 21533.318,E2 21533.318} C_VEL
LIN {X 0,Y 453.465,Z 742.802,A -85,B 0,C 180,E1 21532.083,E2 21532.083} C_VEL
LIN {X 0,Y 452.319,Z 758.317,A -85,B 0,C 180,E1 21530.713,E2 21530.713} C_VEL
LIN {X 0,Y 451.228,Z 773.025,A -85,B 0,C 180,E1 21529.144,E2 21529.144} C_VEL
LIN {X 0,Y 450.276,Z 786.308,A -85,B 0,C 180,E1 21527.444,E2 21527.444} C_VEL
LIN {X 0,Y 449.422,Z 799.025,A -85,B 0,C 180,E1 21525.484,E2 21525.484} C_VEL
LIN {X 0,Y 448.824,Z 810.135,A -85,B 0,C 180,E1 21523.396,E2 21523.396} C_VEL
LIN {X 0,Y 448.398,Z 819.605,A -85,B 0,C 180,E1 21521.186,E2 21521.186} C_VEL
LIN {X 0,Y 448.193,Z 827.057,A -85,B 0,C 180,E1 21518.984,E2 21518.984} C_VEL
LIN {X 0,Y 448.129,Z 832.715,A -85,B 0,C 180,E1 21516.791,E2 21516.791} C_VEL
LIN {X 0,Y 448.121,Z 836.879,A -85,B 0,C 180,E1 21514.479,E2 21514.479} C_VEL
LIN {X 0,Y 448.152,Z 839.283,A -85,B 0,C 180,E1 21512.174,E2 21512.174} C_VEL
LIN {X 0,Y 448.175,Z 839.979,A -85,B 0,C 180,E1 21509.872,E2 21509.872} C_VEL
LIN {X 0,Y 448.156,Z 838.969,A -85,B 0,C 180,E1 21507.571,E2 21507.571} C_VEL
LIN {X 0,Y 448.136,Z 836.23,A -85,B 0,C 180,E1 21505.265,E2 21505.265} C_VEL
LIN {X 0,Y 448.149,Z 831.685,A -85,B 0,C 180,E1 21502.951,E2 21502.951} C_VEL
LIN {X 0,Y 448.222,Z 825.635,A -85,B 0,C 180,E1 21500.758,E2 21500.758} C_VEL
LIN {X 0,Y 448.428,Z 817.69,A -85,B 0,C 180,E1 21498.554,E2 21498.554} C_VEL
LIN {X 0,Y 448.81,Z 808.271,A -85,B 0,C 180,E1 21496.472,E2 21496.472} C_VEL
LIN {X 0,Y 449.373,Z 797.096,A -85,B 0,C 180,E1 21494.457,E2 21494.457} C_VEL
LIN {X 0,Y 450.154,Z 784.281,A -85,B 0,C 180,E1 21492.551,E2 21492.551} C_VEL
LIN {X 0,Y 451.092,Z 769.869,A -85,B 0,C 180,E1 21490.776,E2 21490.776} C_VEL
LIN {X 0,Y 452.191,Z 753.865,A -85,B 0,C 180,E1 21489.145,E2 21489.145} C_VEL
LIN {X 0,Y 453.31,Z 737.463,A -85,B 0,C 180,E1 21487.773,E2 21487.773} C_VEL
LIN {X 0,Y 454.435,Z 720.27,A -85,B 0,C 180,E1 21486.6,E2 21486.6} C_VEL
LIN {X 0,Y 455.513,Z 702.117,A -85,B 0,C 180,E1 21485.628,E2 21485.628} C_VEL
LIN {X 0,Y 456.549,Z 682.542,A -85,B 0,C 180,E1 21484.832,E2 21484.832} C_VEL
LIN {X 0,Y 457.372,Z 662.576,A -85,B 0,C 180,E1 21484.275,E2 21484.275} C_VEL
LIN {X 0,Y 460.267,Z 555.632,A -85,B 0,C 180,E1 21482.145,E2 21482.145} C_VEL
LIN {X 0,Y 462.935,Z 482.739,A -85,B 0,C 180,E1 21480.545,E2 21480.545} C_VEL
LIN {X 0,Y 460.178,Z 455.308,A -85,B 0,C 180,E1 21479.539,E2 21479.539} C_VEL
LIN {X 0,Y 458.973,Z 444.096,A -85,B 0,C 180,E1 21479.061,E2 21479.061} C_VEL
LIN {X 0,Y 461.859,Z 407.041,A -85,B 0,C 180,E1 21475.69,E2 21475.69} C_VEL
LIN {X 0,Y 453.473,Z 383.21,A -85,B 0,C 180,E1 21472.642,E2 21472.642} C_VEL
LIN {X 0,Y 449.071,Z 370.858,A -85,B 0,C 180,E1 21470.942,E2 21470.942} C_VEL
LIN {X 0,Y 449.109,Z 370.858,A -85,B 0,C 180,E1 21467.406,E2 21467.406} C_VEL
LIN {X 0,Y 449.111,Z 370.856,A -85,B 0,C 180,E1 21463.642,E2 21463.642} C_VEL
LIN {X 0,Y 449.076,Z 370.861,A -85,B 0,C 180,E1 21460.012,E2 21460.012} C_VEL
LIN {X 0,Y 449.107,Z 370.867,A -85,B 0,C 180,E1 21457.269,E2 21457.269} C_VEL
LIN {X 0,Y 450.166,Z 374.026,A -85,B 0,C 180,E1 21456.689,E2 21456.689} C_VEL
LIN {X 0,Y 451.794,Z 376.455,A -85,B 0,C 180,E1 21456.12,E2 21456.12} C_VEL
LIN {X 0,Y 455.582,Z 384.404,A -85,B 0,C 180,E1 21454.613,E2 21454.613} C_VEL
LIN {X 0,Y 460.071,Z 395.967,A -85,B 0,C 180,E1 21452.748,E2 21452.748} C_VEL
LIN {X 0,Y 463.258,Z 407.412,A -85,B 0,C 180,E1 21451.162,E2 21451.162} C_VEL
LIN {X 0,Y 463.051,Z 415.236,A -85,B 0,C 180,E1 21450.447,E2 21450.447} C_VEL
LIN {X 0,Y 465.338,Z 429.588,A -85,B 0,C 180,E1 21449.803,E2 21449.803} C_VEL
LIN {X 0,Y 461.101,Z 528.105,A -85,B 0,C 180,E1 21447.648,E2 21447.648} C_VEL
LIN {X 0,Y 458.394,Z 623.148,A -85,B 0,C 180,E1 21445.717,E2 21445.717} C_VEL
LIN {X 0,Y 457.65,Z 642.55,A -85,B 0,C 180,E1 21445.077,E2 21445.077} C_VEL
LIN {X 0,Y 456.759,Z 660.543,A -85,B 0,C 180,E1 21444.256,E2 21444.256} C_VEL
LIN {X 0,Y 455.621,Z 679.164,A -85,B 0,C 180,E1 21443.147,E2 21443.147} C_VEL
LIN {X 0,Y 454.452,Z 695.818,A -85,B 0,C 180,E1 21441.896,E2 21441.896} C_VEL
LIN {X 0,Y 453.267,Z 711.366,A -85,B 0,C 180,E1 21440.465,E2 21440.465} C_VEL
LIN {X 0,Y 452.069,Z 726.215,A -85,B 0,C 180,E1 21438.803,E2 21438.803} C_VEL
LIN {X 0,Y 450.99,Z 739.355,A -85,B 0,C 180,E1 21437.016,E2 21437.016} C_VEL
LIN {X 0,Y 450.048,Z 751.18,A -85,B 0,C 180,E1 21435.066,E2 21435.066} C_VEL
LIN {X 0,Y 449.296,Z 761.474,A -85,B 0,C 180,E1 21432.989,E2 21432.989} C_VEL
LIN {X 0,Y 448.76,Z 769.789,A -85,B 0,C 180,E1 21430.917,E2 21430.917} C_VEL
LIN {X 0,Y 448.39,Z 776.725,A -85,B 0,C 180,E1 21428.721,E2 21428.721} C_VEL
LIN {X 0,Y 448.165,Z 782.188,A -85,B 0,C 180,E1 21426.405,E2 21426.405} C_VEL
LIN {X 0,Y 448.054,Z 785.938,A -85,B 0,C 180,E1 21424.042,E2 21424.042} C_VEL
LIN {X 0,Y 448.015,Z 787.955,A -85,B 0,C 180,E1 21421.662,E2 21421.662} C_VEL
LIN {X 0,Y 448.012,Z 788.237,A -85,B 0,C 180,E1 21419.233,E2 21419.233} C_VEL
LIN {X 0,Y 448.023,Z 786.85,A -85,B 0,C 180,E1 21416.93,E2 21416.93} C_VEL
LIN {X 0,Y 448.078,Z 783.83,A -85,B 0,C 180,E1 21414.622,E2 21414.622} C_VEL
LIN {X 0,Y 448.223,Z 779.098,A -85,B 0,C 180,E1 21412.308,E2 21412.308} C_VEL
LIN {X 0,Y 448.491,Z 772.938,A -85,B 0,C 180,E1 21410.115,E2 21410.115} C_VEL
LIN {X 0,Y 448.947,Z 764.829,A -85,B 0,C 180,E1 21407.88,E2 21407.88} C_VEL
LIN {X 0,Y 449.561,Z 755.566,A -85,B 0,C 180,E1 21405.839,E2 21405.839} C_VEL
LIN {X 0,Y 450.365,Z 744.788,A -85,B 0,C 180,E1 21403.888,E2 21403.888} C_VEL
LIN {X 0,Y 451.343,Z 732.654,A -85,B 0,C 180,E1 21402.065,E2 21402.065} C_VEL
LIN {X 0,Y 452.455,Z 719.13,A -85,B 0,C 180,E1 21400.373,E2 21400.373} C_VEL
LIN {X 0,Y 453.705,Z 703.793,A -85,B 0,C 180,E1 21398.78,E2 21398.78} C_VEL
LIN {X 0,Y 454.966,Z 687.156,A -85,B 0,C 180,E1 21397.372,E2 21397.372} C_VEL
LIN {X 0,Y 456.134,Z 670.182,A -85,B 0,C 180,E1 21396.213,E2 21396.213} C_VEL
LIN {X 0,Y 457.194,Z 652.111,A -85,B 0,C 180,E1 21395.241,E2 21395.241} C_VEL
LIN {X 0,Y 458.074,Z 633.195,A -85,B 0,C 180,E1 21394.477,E2 21394.477} C_VEL
LIN {X 0,Y 458.745,Z 613.549,A -85,B 0,C 180,E1 21393.935,E2 21393.935} C_VEL
LIN {X 0,Y 462.83,Z 427.768,A -85,B 0,C 180,E1 21390.56,E2 21390.56} C_VEL
LIN {X 0,Y 459.279,Z 407.597,A -85,B 0,C 180,E1 21389.88,E2 21389.88} C_VEL
LIN {X 0,Y 459.362,Z 402.642,A -85,B 0,C 180,E1 21389.381,E2 21389.381} C_VEL
LIN {X 0,Y 452.871,Z 382.223,A -85,B 0,C 180,E1 21386.801,E2 21386.801} C_VEL
LIN {X 0,Y 449.072,Z 370.861,A -85,B 0,C 180,E1 21385.289,E2 21385.289} C_VEL
LIN {X 0,Y 449.07,Z 370.859,A -85,B 0,C 180,E1 21381.596,E2 21381.596} C_VEL
LIN {X 0,Y 449.09,Z 370.858,A -85,B 0,C 180,E1 21378.041,E2 21378.041} C_VEL
LIN {X 0,Y 449.117,Z 370.856,A -85,B 0,C 180,E1 21374.351,E2 21374.351} C_VEL
LIN {X 0,Y 449.096,Z 370.856,A -85,B 0,C 180,E1 21372.77,E2 21372.77} C_VEL
LIN {X 0,Y 448.181,Z 370.976,A -85,B 0,C 180,E1 21371.787,E2 21371.787} C_VEL
LIN {X 0,Y 443.446,Z 371.567,A -85,B 0,C 180,E1 21369.866,E2 21369.866} C_VEL
LIN {X 0,Y 441.294,Z 371.831,A -85,B 0,C 180,E1 21368.589,E2 21368.589} C_VEL
LIN {X 0,Y 441.182,Z 371.844,A -85,B 0,C 180,E1 21368.299,E2 21368.299} C_VEL
LIN {X 0,Y 441.177,Z 371.846,A -85,B 0,C 180,E1 21364.416,E2 21364.416} C_VEL
LIN {X 0,Y 441.145,Z 371.846,A -85,B 0,C 180,E1 21360.794,E2 21360.794} C_VEL
LIN {X 0,Y 441.128,Z 371.845,A -85,B 0,C 180,E1 21357.249,E2 21357.249} C_VEL
LIN {X 0,Y 441.132,Z 371.845,A -85,B 0,C 180,E1 21353.511,E2 21353.511} C_VEL
LIN {X 0,Y 441.171,Z 371.846,A -85,B 0,C 180,E1 21350.012,E2 21350.012} C_VEL
LIN {X 0,Y 441.18,Z 371.843,A -85,B 0,C 180,E1 21346.186,E2 21346.186} C_VEL
LIN {X 0,Y 441.144,Z 371.842,A -85,B 0,C 180,E1 21342.567,E2 21342.567} C_VEL
LIN {X 0,Y 441.125,Z 371.842,A -85,B 0,C 180,E1 21338.998,E2 21338.998} C_VEL
LIN {X 0,Y 441.126,Z 371.844,A -85,B 0,C 180,E1 21335.202,E2 21335.202} C_VEL
LIN {X 0,Y 441.145,Z 371.846,A -85,B 0,C 180,E1 21331.559,E2 21331.559} C_VEL
LIN {X 0,Y 441.175,Z 371.84,A -85,B 0,C 180,E1 21327.922,E2 21327.922} C_VEL
LIN {X 0,Y 441.163,Z 371.845,A -85,B 0,C 180,E1 21324.146,E2 21324.146} C_VEL
LIN {X 0,Y 441.129,Z 371.844,A -85,B 0,C 180,E1 21320.608,E2 21320.608} C_VEL
LIN {X 0,Y 441.124,Z 371.844,A -85,B 0,C 180,E1 21316.899,E2 21316.899} C_VEL
LIN {X 0,Y 441.141,Z 371.845,A -85,B 0,C 180,E1 21313.271,E2 21313.271} C_VEL
LIN {X 0,Y 441.169,Z 371.845,A -85,B 0,C 180,E1 21309.572,E2 21309.572} C_VEL
LIN {X 0,Y 441.163,Z 371.845,A -85,B 0,C 180,E1 21305.923,E2 21305.923} C_VEL
LIN {X 0,Y 441.133,Z 371.845,A -85,B 0,C 180,E1 21302.312,E2 21302.312} C_VEL
LIN {X 0,Y 441.124,Z 371.847,A -85,B 0,C 180,E1 21298.707,E2 21298.707} C_VEL
LIN {X 0,Y 441.135,Z 371.85,A -85,B 0,C 180,E1 21295.009,E2 21295.009} C_VEL
LIN {X 0,Y 441.178,Z 371.848,A -85,B 0,C 180,E1 21291.434,E2 21291.434} C_VEL
LIN {X 0,Y 441.172,Z 371.846,A -85,B 0,C 180,E1 21287.633,E2 21287.633} C_VEL
LIN {X 0,Y 441.146,Z 371.847,A -85,B 0,C 180,E1 21283.883,E2 21283.883} C_VEL
LIN {X 0,Y 441.125,Z 371.849,A -85,B 0,C 180,E1 21280.24,E2 21280.24} C_VEL
LIN {X 0,Y 441.122,Z 371.85,A -85,B 0,C 180,E1 21276.423,E2 21276.423} C_VEL
LIN {X 0,Y 441.148,Z 371.98,A -85,B 0,C 180,E1 21274.022,E2 21274.022} C_VEL
LIN {X 0,Y 446.56,Z 391.743,A -85,B 0,C 180,E1 21270.697,E2 21270.697} C_VEL
LIN {X 0,Y 448.694,Z 400.538,A -85,B 0,C 180,E1 21269.284,E2 21269.284} C_VEL
LIN {X 0,Y 446.856,Z 427.964,A -85,B 0,C 180,E1 21265.514,E2 21265.514} C_VEL
LIN {X 0,Y 445.149,Z 456.259,A -85,B 0,C 180,E1 21261.684,E2 21261.684} C_VEL
LIN {X 0,Y 444.007,Z 479.54,A -85,B 0,C 180,E1 21258.616,E2 21258.616} C_VEL
LIN {X 0,Y 446.845,Z 499.932,A -85,B 0,C 180,E1 21258.054,E2 21258.054} C_VEL
LIN {X 0,Y 444.857,Z 600.58,A -85,B 0,C 180,E1 21256.049,E2 21256.049} C_VEL
LIN {X 0,Y 444.511,Z 616.268,A -85,B 0,C 180,E1 21255.498,E2 21255.498} C_VEL
LIN {X 0,Y 444.053,Z 631.04,A -85,B 0,C 180,E1 21254.74,E2 21254.74} C_VEL
LIN {X 0,Y 443.456,Z 645.186,A -85,B 0,C 180,E1 21253.761,E2 21253.761} C_VEL
LIN {X 0,Y 442.897,Z 657.682,A -85,B 0,C 180,E1 21252.649,E2 21252.649} C_VEL
LIN {X 0,Y 442.349,Z 669.883,A -85,B 0,C 180,E1 21251.275,E2 21251.275} C_VEL
LIN {X 0,Y 441.843,Z 680.376,A -85,B 0,C 180,E1 21249.772,E2 21249.772} C_VEL
LIN {X 0,Y 441.466,Z 689.052,A -85,B 0,C 180,E1 21248.204,E2 21248.204} C_VEL
LIN {X 0,Y 441.163,Z 696.839,A -85,B 0,C 180,E1 21246.376,E2 21246.376} C_VEL
LIN {X 0,Y 440.981,Z 702.817,A -85,B 0,C 180,E1 21244.421,E2 21244.421} C_VEL
LIN {X 0,Y 440.905,Z 706.498,A -85,B 0,C 180,E1 21242.6,E2 21242.6} C_VEL
LIN {X 0,Y 440.931,Z 708.61,A -85,B 0,C 180,E1 21240.65,E2 21240.65} C_VEL
LIN {X 0,Y 440.996,Z 708.804,A -85,B 0,C 180,E1 21238.701,E2 21238.701} C_VEL
LIN {X 0,Y 441.149,Z 707.31,A -85,B 0,C 180,E1 21236.882,E2 21236.882} C_VEL
LIN {X 0,Y 441.394,Z 703.804,A -85,B 0,C 180,E1 21234.932,E2 21234.932} C_VEL
LIN {X 0,Y 441.743,Z 698.588,A -85,B 0,C 180,E1 21233.11,E2 21233.11} C_VEL
LIN {X 0,Y 442.185,Z 691.922,A -85,B 0,C 180,E1 21231.417,E2 21231.417} C_VEL
LIN {X 0,Y 442.76,Z 683.09,A -85,B 0,C 180,E1 21229.724,E2 21229.724} C_VEL
LIN {X 0,Y 443.418,Z 673.03,A -85,B 0,C 180,E1 21228.225,E2 21228.225} C_VEL
LIN {X 0,Y 444.131,Z 661.415,A -85,B 0,C 180,E1 21226.857,E2 21226.857} C_VEL
LIN {X 0,Y 444.86,Z 648.066,A -85,B 0,C 180,E1 21225.63,E2 21225.63} C_VEL
LIN {X 0,Y 445.617,Z 633.218,A -85,B 0,C 180,E1 21224.581,E2 21224.581} C_VEL
LIN {X 0,Y 446.208,Z 618.421,A -85,B 0,C 180,E1 21223.801,E2 21223.801} C_VEL
LIN {X 0,Y 446.703,Z 602.508,A -85,B 0,C 180,E1 21223.213,E2 21223.213} C_VEL
LIN {X 0,Y 450.882,Z 507.375,A -85,B 0,C 180,E1 21220.757,E2 21220.757} C_VEL
LIN {X 0,Y 451.034,Z 500.084,A -85,B 0,C 180,E1 21220.543,E2 21220.543} C_VEL
LIN {X 0,Y 447.265,Z 479.204,A -85,B 0,C 180,E1 21219.556,E2 21219.556} C_VEL
LIN {X 0,Y 449.897,Z 451.736,A -85,B 0,C 180,E1 21215.583,E2 21215.583} C_VEL
LIN {X 0,Y 453.131,Z 425.938,A -85,B 0,C 180,E1 21211.679,E2 21211.679} C_VEL
LIN {X 0,Y 455.183,Z 411.883,A -85,B 0,C 180,E1 21209.438,E2 21209.438} C_VEL
LIN {X 0,Y 453.06,Z 402.387,A -85,B 0,C 180,E1 21207.228,E2 21207.228} C_VEL
LIN {X 0,Y 450.849,Z 394.904,A -85,B 0,C 180,E1 21205.098,E2 21205.098} C_VEL
LIN {X 0,Y 448.742,Z 388.733,A -85,B 0,C 180,E1 21202.856,E2 21202.856} C_VEL
LIN {X 0,Y 447.259,Z 384.999,A -85,B 0,C 180,E1 21200.919,E2 21200.919} C_VEL
LIN {X 0,Y 446.194,Z 382.233,A -85,B 0,C 180,E1 21198.448,E2 21198.448} C_VEL
LIN {X 0,Y 446.244,Z 381.669,A -85,B 0,C 180,E1 21196.361,E2 21196.361} C_VEL
LIN {X 0,Y 446.66,Z 383.485,A -85,B 0,C 180,E1 21194.248,E2 21194.248} C_VEL
